Fanuc TP program (LS listing): FM144712.ls

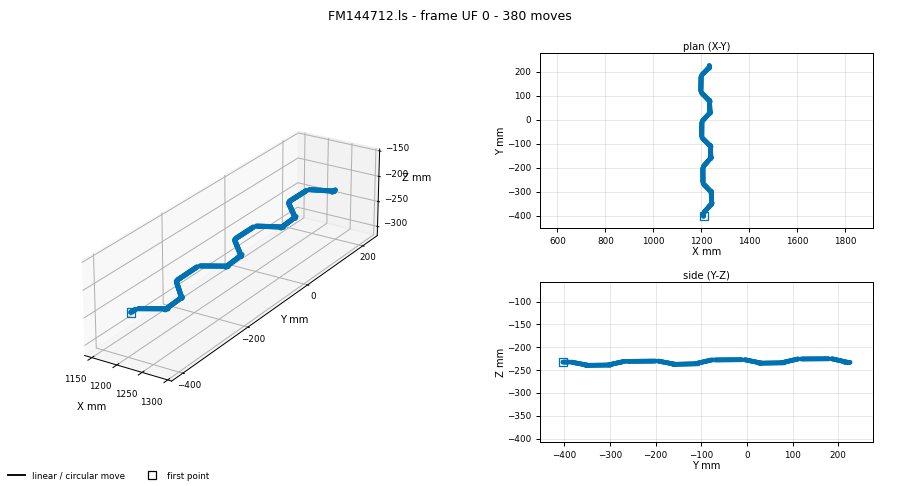
[picture p0: tool path of FM144712.ls in frame UF 0, 380 of 380 moves have a stored position in this frame; points joined in program order, loops and branches not executed]
/PROG  FM144712
/ATTR
OWNER		= MNEDITOR;
COMMENT		= "Auto FANUC move";
PROG_SIZE	= 0;
CREATE		= DATE 26-05-06  TIME 14:47:12;
MODIFIED	= DATE 26-05-06  TIME 14:47:12;
FILE_NAME	= ;
VERSION		= 0;
LINE_COUNT	= 385;
MEMORY_SIZE	= 0;
PROTECT		= READ_WRITE;
TCD:  STACK_SIZE	= 0,
      TASK_PRIORITY	= 50,
      TIME_SLICE	= 0,
      BUSY_LAMP_OFF	= 0,
      ABORT_REQUEST	= 0,
      PAUSE_REQUEST	= 0;
DEFAULT_GROUP	= 1,*,*,*,*;
CONTROL_CODE	= 00000000 00000000;
/MN
   1:  UFRAME_NUM=0 ;
   2:  UTOOL_NUM=1 ;
   3:  R[93]=10 ;
   4:  L P[1] 7mm/sec FINE ;
   5:  L P[2] 7mm/sec CNT50 ;
   6:  L P[3] 7mm/sec CNT50 ;
   7:  L P[4] 7mm/sec CNT50 ;
   8:  L P[5] 7mm/sec CNT50 ;
   9:  L P[6] 7mm/sec CNT50 ;
  10:  L P[7] 7mm/sec CNT50 ;
  11:  L P[8] 7mm/sec CNT50 ;
  12:  L P[9] 7mm/sec CNT50 ;
  13:  L P[10] 7mm/sec CNT50 ;
  14:  L P[11] 7mm/sec CNT50 ;
  15:  L P[12] 7mm/sec CNT50 ;
  16:  L P[13] 7mm/sec CNT50 ;
  17:  L P[14] 7mm/sec CNT50 ;
  18:  L P[15] 7mm/sec CNT50 ;
  19:  L P[16] 7mm/sec CNT50 ;
  20:  L P[17] 7mm/sec CNT50 ;
  21:  L P[18] 7mm/sec CNT50 ;
  22:  L P[19] 7mm/sec CNT50 ;
  23:  L P[20] 7mm/sec CNT50 ;
  24:  L P[21] 7mm/sec CNT50 ;
  25:  L P[22] 7mm/sec CNT50 ;
  26:  L P[23] 7mm/sec CNT50 ;
  27:  L P[24] 7mm/sec CNT50 ;
  28:  L P[25] 7mm/sec CNT50 ;
  29:  L P[26] 7mm/sec CNT50 ;
  30:  L P[27] 7mm/sec CNT50 ;
  31:  L P[28] 7mm/sec CNT50 ;
  32:  L P[29] 7mm/sec CNT50 ;
  33:  L P[30] 7mm/sec CNT50 ;
  34:  L P[31] 7mm/sec CNT50 ;
  35:  L P[32] 7mm/sec CNT50 ;
  36:  L P[33] 7mm/sec CNT50 ;
  37:  L P[34] 7mm/sec CNT50 ;
  38:  L P[35] 7mm/sec CNT50 ;
  39:  L P[36] 7mm/sec CNT50 ;
  40:  L P[37] 7mm/sec CNT50 ;
  41:  L P[38] 7mm/sec CNT50 ;
  42:  L P[39] 7mm/sec CNT50 ;
  43:  L P[40] 7mm/sec CNT50 ;
  44:  L P[41] 7mm/sec CNT50 ;
  45:  L P[42] 7mm/sec CNT50 ;
  46:  L P[43] 7mm/sec CNT50 ;
  47:  L P[44] 7mm/sec CNT50 ;
  48:  L P[45] 7mm/sec CNT50 ;
  49:  L P[46] 7mm/sec CNT50 ;
  50:  L P[47] 7mm/sec CNT50 ;
  51:  L P[48] 7mm/sec CNT50 ;
  52:  L P[49] 7mm/sec CNT50 ;
  53:  L P[50] 7mm/sec CNT50 ;
  54:  L P[51] 7mm/sec CNT50 ;
  55:  L P[52] 7mm/sec CNT50 ;
  56:  L P[53] 7mm/sec CNT50 ;
  57:  L P[54] 7mm/sec CNT50 ;
  58:  L P[55] 7mm/sec CNT50 ;
  59:  L P[56] 7mm/sec CNT50 ;
  60:  L P[57] 7mm/sec CNT50 ;
  61:  L P[58] 7mm/sec CNT50 ;
  62:  L P[59] 7mm/sec CNT50 ;
  63:  L P[60] 7mm/sec CNT50 ;
  64:  L P[61] 7mm/sec CNT50 ;
  65:  L P[62] 7mm/sec CNT50 ;
  66:  L P[63] 7mm/sec CNT50 ;
  67:  L P[64] 7mm/sec CNT50 ;
  68:  L P[65] 7mm/sec CNT50 ;
  69:  L P[66] 7mm/sec CNT50 ;
  70:  L P[67] 7mm/sec CNT50 ;
  71:  L P[68] 7mm/sec CNT50 ;
  72:  L P[69] 7mm/sec CNT50 ;
  73:  L P[70] 7mm/sec CNT50 ;
  74:  L P[71] 7mm/sec CNT50 ;
  75:  L P[72] 7mm/sec CNT50 ;
  76:  L P[73] 7mm/sec CNT50 ;
  77:  L P[74] 7mm/sec CNT50 ;
  78:  L P[75] 7mm/sec CNT50 ;
  79:  L P[76] 7mm/sec CNT50 ;
  80:  L P[77] 7mm/sec CNT50 ;
  81:  L P[78] 7mm/sec CNT50 ;
  82:  L P[79] 7mm/sec CNT50 ;
  83:  L P[80] 7mm/sec CNT50 ;
  84:  L P[81] 7mm/sec CNT50 ;
  85:  L P[82] 7mm/sec CNT50 ;
  86:  L P[83] 7mm/sec CNT50 ;
  87:  L P[84] 7mm/sec CNT50 ;
  88:  L P[85] 7mm/sec CNT50 ;
  89:  L P[86] 7mm/sec CNT50 ;
  90:  L P[87] 7mm/sec CNT50 ;
  91:  L P[88] 7mm/sec CNT50 ;
  92:  L P[89] 7mm/sec CNT50 ;
  93:  L P[90] 7mm/sec CNT50 ;
  94:  L P[91] 7mm/sec CNT50 ;
  95:  L P[92] 7mm/sec CNT50 ;
  96:  L P[93] 7mm/sec CNT50 ;
  97:  L P[94] 7mm/sec CNT50 ;
  98:  L P[95] 7mm/sec CNT50 ;
  99:  L P[96] 7mm/sec CNT50 ;
 100:  L P[97] 7mm/sec CNT50 ;
 101:  L P[98] 7mm/sec CNT50 ;
 102:  L P[99] 7mm/sec CNT50 ;
 103:  L P[100] 7mm/sec CNT50 ;
 104:  L P[101] 7mm/sec CNT50 ;
 105:  L P[102] 7mm/sec CNT50 ;
 106:  L P[103] 7mm/sec CNT50 ;
 107:  L P[104] 7mm/sec CNT50 ;
 108:  L P[105] 7mm/sec CNT50 ;
 109:  L P[106] 7mm/sec CNT50 ;
 110:  L P[107] 7mm/sec CNT50 ;
 111:  L P[108] 7mm/sec CNT50 ;
 112:  L P[109] 7mm/sec CNT50 ;
 113:  L P[110] 7mm/sec CNT50 ;
 114:  L P[111] 7mm/sec CNT50 ;
 115:  L P[112] 7mm/sec CNT50 ;
 116:  L P[113] 7mm/sec CNT50 ;
 117:  L P[114] 7mm/sec CNT50 ;
 118:  L P[115] 7mm/sec CNT50 ;
 119:  L P[116] 7mm/sec CNT50 ;
 120:  L P[117] 7mm/sec CNT50 ;
 121:  L P[118] 7mm/sec CNT50 ;
 122:  L P[119] 7mm/sec CNT50 ;
 123:  L P[120] 7mm/sec CNT50 ;
 124:  L P[121] 7mm/sec CNT50 ;
 125:  L P[122] 7mm/sec CNT50 ;
 126:  L P[123] 7mm/sec CNT50 ;
 127:  L P[124] 7mm/sec CNT50 ;
 128:  L P[125] 7mm/sec CNT50 ;
 129:  L P[126] 7mm/sec CNT50 ;
 130:  L P[127] 7mm/sec CNT50 ;
 131:  L P[128] 7mm/sec CNT50 ;
 132:  L P[129] 7mm/sec CNT50 ;
 133:  L P[130] 7mm/sec CNT50 ;
 134:  L P[131] 7mm/sec CNT50 ;
 135:  L P[132] 7mm/sec CNT50 ;
 136:  L P[133] 7mm/sec CNT50 ;
 137:  L P[134] 7mm/sec CNT50 ;
 138:  L P[135] 7mm/sec CNT50 ;
 139:  L P[136] 7mm/sec CNT50 ;
 140:  L P[137] 7mm/sec CNT50 ;
 141:  L P[138] 7mm/sec CNT50 ;
 142:  L P[139] 7mm/sec CNT50 ;
 143:  L P[140] 7mm/sec CNT50 ;
 144:  L P[141] 7mm/sec CNT50 ;
 145:  L P[142] 7mm/sec CNT50 ;
 146:  L P[143] 7mm/sec CNT50 ;
 147:  L P[144] 7mm/sec CNT50 ;
 148:  L P[145] 7mm/sec CNT50 ;
 149:  L P[146] 7mm/sec CNT50 ;
 150:  L P[147] 7mm/sec CNT50 ;
 151:  L P[148] 7mm/sec CNT50 ;
 152:  L P[149] 7mm/sec CNT50 ;
 153:  L P[150] 7mm/sec CNT50 ;
 154:  L P[151] 7mm/sec CNT50 ;
 155:  L P[152] 7mm/sec CNT50 ;
 156:  L P[153] 7mm/sec CNT50 ;
 157:  L P[154] 7mm/sec CNT50 ;
 158:  L P[155] 7mm/sec CNT50 ;
 159:  L P[156] 7mm/sec CNT50 ;
 160:  L P[157] 7mm/sec CNT50 ;
 161:  L P[158] 7mm/sec CNT50 ;
 162:  L P[159] 7mm/sec CNT50 ;
 163:  L P[160] 7mm/sec CNT50 ;
 164:  L P[161] 7mm/sec CNT50 ;
 165:  L P[162] 7mm/sec CNT50 ;
 166:  L P[163] 7mm/sec CNT50 ;
 167:  L P[164] 7mm/sec CNT50 ;
 168:  L P[165] 7mm/sec CNT50 ;
 169:  L P[166] 7mm/sec CNT50 ;
 170:  L P[167] 7mm/sec CNT50 ;
 171:  L P[168] 7mm/sec CNT50 ;
 172:  L P[169] 7mm/sec CNT50 ;
 173:  L P[170] 7mm/sec CNT50 ;
 174:  L P[171] 7mm/sec CNT50 ;
 175:  L P[172] 7mm/sec CNT50 ;
 176:  L P[173] 7mm/sec CNT50 ;
 177:  L P[174] 7mm/sec CNT50 ;
 178:  L P[175] 7mm/sec CNT50 ;
 179:  L P[176] 7mm/sec CNT50 ;
 180:  L P[177] 7mm/sec CNT50 ;
 181:  L P[178] 7mm/sec CNT50 ;
 182:  L P[179] 7mm/sec CNT50 ;
 183:  L P[180] 7mm/sec CNT50 ;
 184:  L P[181] 7mm/sec CNT50 ;
 185:  L P[182] 7mm/sec CNT50 ;
 186:  L P[183] 7mm/sec CNT50 ;
 187:  L P[184] 7mm/sec CNT50 ;
 188:  L P[185] 7mm/sec CNT50 ;
 189:  L P[186] 7mm/sec CNT50 ;
 190:  L P[187] 7mm/sec CNT50 ;
 191:  L P[188] 7mm/sec CNT50 ;
 192:  L P[189] 7mm/sec CNT50 ;
 193:  L P[190] 7mm/sec CNT50 ;
 194:  L P[191] 7mm/sec CNT50 ;
 195:  L P[192] 7mm/sec CNT50 ;
 196:  L P[193] 7mm/sec CNT50 ;
 197:  L P[194] 7mm/sec CNT50 ;
 198:  L P[195] 7mm/sec CNT50 ;
 199:  L P[196] 7mm/sec CNT50 ;
 200:  L P[197] 7mm/sec CNT50 ;
 201:  L P[198] 7mm/sec CNT50 ;
 202:  L P[199] 7mm/sec CNT50 ;
 203:  L P[200] 7mm/sec CNT50 ;
 204:  L P[201] 7mm/sec CNT50 ;
 205:  L P[202] 7mm/sec CNT50 ;
 206:  L P[203] 7mm/sec CNT50 ;
 207:  L P[204] 7mm/sec CNT50 ;
 208:  L P[205] 7mm/sec CNT50 ;
 209:  L P[206] 7mm/sec CNT50 ;
 210:  L P[207] 7mm/sec CNT50 ;
 211:  L P[208] 7mm/sec CNT50 ;
 212:  L P[209] 7mm/sec CNT50 ;
 213:  L P[210] 7mm/sec CNT50 ;
 214:  L P[211] 7mm/sec CNT50 ;
 215:  L P[212] 7mm/sec CNT50 ;
 216:  L P[213] 7mm/sec CNT50 ;
 217:  L P[214] 7mm/sec CNT50 ;
 218:  L P[215] 7mm/sec CNT50 ;
 219:  L P[216] 7mm/sec CNT50 ;
 220:  L P[217] 7mm/sec CNT50 ;
 221:  L P[218] 7mm/sec CNT50 ;
 222:  L P[219] 7mm/sec CNT50 ;
 223:  L P[220] 7mm/sec CNT50 ;
 224:  L P[221] 7mm/sec CNT50 ;
 225:  L P[222] 7mm/sec CNT50 ;
 226:  L P[223] 7mm/sec CNT50 ;
 227:  L P[224] 7mm/sec CNT50 ;
 228:  L P[225] 7mm/sec CNT50 ;
 229:  L P[226] 7mm/sec CNT50 ;
 230:  L P[227] 7mm/sec CNT50 ;
 231:  L P[228] 7mm/sec CNT50 ;
 232:  L P[229] 7mm/sec CNT50 ;
 233:  L P[230] 7mm/sec CNT50 ;
 234:  L P[231] 7mm/sec CNT50 ;
 235:  L P[232] 7mm/sec CNT50 ;
 236:  L P[233] 7mm/sec CNT50 ;
 237:  L P[234] 7mm/sec CNT50 ;
 238:  L P[235] 7mm/sec CNT50 ;
 239:  L P[236] 7mm/sec CNT50 ;
 240:  L P[237] 7mm/sec CNT50 ;
 241:  L P[238] 7mm/sec CNT50 ;
 242:  L P[239] 7mm/sec CNT50 ;
 243:  L P[240] 7mm/sec CNT50 ;
 244:  L P[241] 7mm/sec CNT50 ;
 245:  L P[242] 7mm/sec CNT50 ;
 246:  L P[243] 7mm/sec CNT50 ;
 247:  L P[244] 7mm/sec CNT50 ;
 248:  L P[245] 7mm/sec CNT50 ;
 249:  L P[246] 7mm/sec CNT50 ;
 250:  L P[247] 7mm/sec CNT50 ;
 251:  L P[248] 7mm/sec CNT50 ;
 252:  L P[249] 7mm/sec CNT50 ;
 253:  L P[250] 7mm/sec CNT50 ;
 254:  L P[251] 7mm/sec CNT50 ;
 255:  L P[252] 7mm/sec CNT50 ;
 256:  L P[253] 7mm/sec CNT50 ;
 257:  L P[254] 7mm/sec CNT50 ;
 258:  L P[255] 7mm/sec CNT50 ;
 259:  L P[256] 7mm/sec CNT50 ;
 260:  L P[257] 7mm/sec CNT50 ;
 261:  L P[258] 7mm/sec CNT50 ;
 262:  L P[259] 7mm/sec CNT50 ;
 263:  L P[260] 7mm/sec CNT50 ;
 264:  L P[261] 7mm/sec CNT50 ;
 265:  L P[262] 7mm/sec CNT50 ;
 266:  L P[263] 7mm/sec CNT50 ;
 267:  L P[264] 7mm/sec CNT50 ;
 268:  L P[265] 7mm/sec CNT50 ;
 269:  L P[266] 7mm/sec CNT50 ;
 270:  L P[267] 7mm/sec CNT50 ;
 271:  L P[268] 7mm/sec CNT50 ;
 272:  L P[269] 7mm/sec CNT50 ;
 273:  L P[270] 7mm/sec CNT50 ;
 274:  L P[271] 7mm/sec CNT50 ;
 275:  L P[272] 7mm/sec CNT50 ;
 276:  L P[273] 7mm/sec CNT50 ;
 277:  L P[274] 7mm/sec CNT50 ;
 278:  L P[275] 7mm/sec CNT50 ;
 279:  L P[276] 7mm/sec CNT50 ;
 280:  L P[277] 7mm/sec CNT50 ;
 281:  L P[278] 7mm/sec CNT50 ;
 282:  L P[279] 7mm/sec CNT50 ;
 283:  L P[280] 7mm/sec CNT50 ;
 284:  L P[281] 7mm/sec CNT50 ;
 285:  L P[282] 7mm/sec CNT50 ;
 286:  L P[283] 7mm/sec CNT50 ;
 287:  L P[284] 7mm/sec CNT50 ;
 288:  L P[285] 7mm/sec CNT50 ;
 289:  L P[286] 7mm/sec CNT50 ;
 290:  L P[287] 7mm/sec CNT50 ;
 291:  L P[288] 7mm/sec CNT50 ;
 292:  L P[289] 7mm/sec CNT50 ;
 293:  L P[290] 7mm/sec CNT50 ;
 294:  L P[291] 7mm/sec CNT50 ;
 295:  L P[292] 7mm/sec CNT50 ;
 296:  L P[293] 7mm/sec CNT50 ;
 297:  L P[294] 7mm/sec CNT50 ;
 298:  L P[295] 7mm/sec CNT50 ;
 299:  L P[296] 7mm/sec CNT50 ;
 300:  L P[297] 7mm/sec CNT50 ;
 301:  L P[298] 7mm/sec CNT50 ;
 302:  L P[299] 7mm/sec CNT50 ;
 303:  L P[300] 7mm/sec CNT50 ;
 304:  L P[301] 7mm/sec CNT50 ;
 305:  L P[302] 7mm/sec CNT50 ;
 306:  L P[303] 7mm/sec CNT50 ;
 307:  L P[304] 7mm/sec CNT50 ;
 308:  L P[305] 7mm/sec CNT50 ;
 309:  L P[306] 7mm/sec CNT50 ;
 310:  L P[307] 7mm/sec CNT50 ;
 311:  L P[308] 7mm/sec CNT50 ;
 312:  L P[309] 7mm/sec CNT50 ;
 313:  L P[310] 7mm/sec CNT50 ;
 314:  L P[311] 7mm/sec CNT50 ;
 315:  L P[312] 7mm/sec CNT50 ;
 316:  L P[313] 7mm/sec CNT50 ;
 317:  L P[314] 7mm/sec CNT50 ;
 318:  L P[315] 7mm/sec CNT50 ;
 319:  L P[316] 7mm/sec CNT50 ;
 320:  L P[317] 7mm/sec CNT50 ;
 321:  L P[318] 7mm/sec CNT50 ;
 322:  L P[319] 7mm/sec CNT50 ;
 323:  L P[320] 7mm/sec CNT50 ;
 324:  L P[321] 7mm/sec CNT50 ;
 325:  L P[322] 7mm/sec CNT50 ;
 326:  L P[323] 7mm/sec CNT50 ;
 327:  L P[324] 7mm/sec CNT50 ;
 328:  L P[325] 7mm/sec CNT50 ;
 329:  L P[326] 7mm/sec CNT50 ;
 330:  L P[327] 7mm/sec CNT50 ;
 331:  L P[328] 7mm/sec CNT50 ;
 332:  L P[329] 7mm/sec CNT50 ;
 333:  L P[330] 7mm/sec CNT50 ;
 334:  L P[331] 7mm/sec CNT50 ;
 335:  L P[332] 7mm/sec CNT50 ;
 336:  L P[333] 7mm/sec CNT50 ;
 337:  L P[334] 7mm/sec CNT50 ;
 338:  L P[335] 7mm/sec CNT50 ;
 339:  L P[336] 7mm/sec CNT50 ;
 340:  L P[337] 7mm/sec CNT50 ;
 341:  L P[338] 7mm/sec CNT50 ;
 342:  L P[339] 7mm/sec CNT50 ;
 343:  L P[340] 7mm/sec CNT50 ;
 344:  L P[341] 7mm/sec CNT50 ;
 345:  L P[342] 7mm/sec CNT50 ;
 346:  L P[343] 7mm/sec CNT50 ;
 347:  L P[344] 7mm/sec CNT50 ;
 348:  L P[345] 7mm/sec CNT50 ;
 349:  L P[346] 7mm/sec CNT50 ;
 350:  L P[347] 7mm/sec CNT50 ;
 351:  L P[348] 7mm/sec CNT50 ;
 352:  L P[349] 7mm/sec CNT50 ;
 353:  L P[350] 7mm/sec CNT50 ;
 354:  L P[351] 7mm/sec CNT50 ;
 355:  L P[352] 7mm/sec CNT50 ;
 356:  L P[353] 7mm/sec CNT50 ;
 357:  L P[354] 7mm/sec CNT50 ;
 358:  L P[355] 7mm/sec CNT50 ;
 359:  L P[356] 7mm/sec CNT50 ;
 360:  L P[357] 7mm/sec CNT50 ;
 361:  L P[358] 7mm/sec CNT50 ;
 362:  L P[359] 7mm/sec CNT50 ;
 363:  L P[360] 7mm/sec CNT50 ;
 364:  L P[361] 7mm/sec CNT50 ;
 365:  L P[362] 7mm/sec CNT50 ;
 366:  L P[363] 7mm/sec CNT50 ;
 367:  L P[364] 7mm/sec CNT50 ;
 368:  L P[365] 7mm/sec CNT50 ;
 369:  L P[366] 7mm/sec CNT50 ;
 370:  L P[367] 7mm/sec CNT50 ;
 371:  L P[368] 7mm/sec CNT50 ;
 372:  L P[369] 7mm/sec CNT50 ;
 373:  L P[370] 7mm/sec CNT50 ;
 374:  L P[371] 7mm/sec CNT50 ;
 375:  L P[372] 7mm/sec CNT50 ;
 376:  L P[373] 7mm/sec CNT50 ;
 377:  L P[374] 7mm/sec CNT50 ;
 378:  L P[375] 7mm/sec CNT50 ;
 379:  L P[376] 7mm/sec CNT50 ;
 380:  L P[377] 7mm/sec CNT50 ;
 381:  L P[378] 7mm/sec CNT50 ;
 382:  L P[379] 7mm/sec CNT50 ;
 383:  L P[380] 7mm/sec FINE ;
 384:  R[93]=1 ;
 385:  END ;
/POS
P[1]{
   GP1:
	UF : 0, UT : 1,		CONFIG : 'N U T, 0, 0, 0',
	X = 1209.451  mm,	Y = -403.216  mm,	Z = -232.520  mm,
	W = 0.000 deg,	P = 30.000 deg,	R = 178.127 deg
};
P[2]{
   GP1:
	UF : 0, UT : 1,		CONFIG : 'N U T, 0, 0, 0',
	X = 1209.517  mm,	Y = -401.217  mm,	Z = -232.512  mm,
	W = 0.000 deg,	P = 30.000 deg,	R = 178.127 deg
};
P[3]{
   GP1:
	UF : 0, UT : 1,		CONFIG : 'N U T, 0, 0, 0',
	X = 1209.582  mm,	Y = -399.218  mm,	Z = -232.503  mm,
	W = 0.000 deg,	P = 30.000 deg,	R = 170.876 deg
};
P[4]{
   GP1:
	UF : 0, UT : 1,		CONFIG : 'N U T, 0, 0, 0',
	X = 1209.647  mm,	Y = -397.220  mm,	Z = -232.495  mm,
	W = 0.000 deg,	P = 30.000 deg,	R = 167.251 deg
};
P[5]{
   GP1:
	UF : 0, UT : 1,		CONFIG : 'N U T, 0, 0, 0',
	X = 1209.713  mm,	Y = -395.221  mm,	Z = -232.486  mm,
	W = 0.000 deg,	P = 30.000 deg,	R = 163.625 deg
};
P[6]{
   GP1:
	UF : 0, UT : 1,		CONFIG : 'N U T, 0, 0, 0',
	X = 1209.778  mm,	Y = -393.222  mm,	Z = -232.478  mm,
	W = 0.000 deg,	P = 30.000 deg,	R = 160.000 deg
};
P[7]{
   GP1:
	UF : 0, UT : 1,		CONFIG : 'N U T, 0, 0, 0',
	X = 1209.922  mm,	Y = -390.499  mm,	Z = -232.471  mm,
	W = 0.000 deg,	P = 30.000 deg,	R = 160.000 deg
};
P[8]{
   GP1:
	UF : 0, UT : 1,		CONFIG : 'N U T, 0, 0, 0',
	X = 1212.525  mm,	Y = -385.034  mm,	Z = -232.516  mm,
	W = 0.000 deg,	P = 30.000 deg,	R = 160.000 deg
};
P[9]{
   GP1:
	UF : 0, UT : 1,		CONFIG : 'N U T, 0, 0, 0',
	X = 1213.831  mm,	Y = -383.546  mm,	Z = -232.798  mm,
	W = 0.000 deg,	P = 30.000 deg,	R = 160.000 deg
};
P[10]{
   GP1:
	UF : 0, UT : 1,		CONFIG : 'N U T, 0, 0, 0',
	X = 1215.138  mm,	Y = -382.058  mm,	Z = -233.080  mm,
	W = 0.000 deg,	P = 30.000 deg,	R = 160.000 deg
};
P[11]{
   GP1:
	UF : 0, UT : 1,		CONFIG : 'N U T, 0, 0, 0',
	X = 1216.444  mm,	Y = -380.570  mm,	Z = -233.362  mm,
	W = 0.000 deg,	P = 30.000 deg,	R = 160.000 deg
};
P[12]{
   GP1:
	UF : 0, UT : 1,		CONFIG : 'N U T, 0, 0, 0',
	X = 1217.751  mm,	Y = -379.082  mm,	Z = -233.644  mm,
	W = 0.000 deg,	P = 30.000 deg,	R = 160.000 deg
};
P[13]{
   GP1:
	UF : 0, UT : 1,		CONFIG : 'N U T, 0, 0, 0',
	X = 1219.057  mm,	Y = -377.595  mm,	Z = -233.926  mm,
	W = 0.000 deg,	P = 30.000 deg,	R = 160.000 deg
};
P[14]{
   GP1:
	UF : 0, UT : 1,		CONFIG : 'N U T, 0, 0, 0',
	X = 1220.364  mm,	Y = -376.107  mm,	Z = -234.208  mm,
	W = 0.000 deg,	P = 30.000 deg,	R = 160.000 deg
};
P[15]{
   GP1:
	UF : 0, UT : 1,		CONFIG : 'N U T, 0, 0, 0',
	X = 1221.670  mm,	Y = -374.619  mm,	Z = -234.490  mm,
	W = 0.000 deg,	P = 30.000 deg,	R = 160.000 deg
};
P[16]{
   GP1:
	UF : 0, UT : 1,		CONFIG : 'N U T, 0, 0, 0',
	X = 1222.977  mm,	Y = -373.131  mm,	Z = -234.772  mm,
	W = 0.000 deg,	P = 30.000 deg,	R = 160.000 deg
};
P[17]{
   GP1:
	UF : 0, UT : 1,		CONFIG : 'N U T, 0, 0, 0',
	X = 1224.283  mm,	Y = -371.644  mm,	Z = -235.054  mm,
	W = 0.000 deg,	P = 30.000 deg,	R = 160.000 deg
};
P[18]{
   GP1:
	UF : 0, UT : 1,		CONFIG : 'N U T, 0, 0, 0',
	X = 1225.590  mm,	Y = -370.156  mm,	Z = -235.336  mm,
	W = 0.000 deg,	P = 30.000 deg,	R = 160.000 deg
};
P[19]{
   GP1:
	UF : 0, UT : 1,		CONFIG : 'N U T, 0, 0, 0',
	X = 1226.896  mm,	Y = -368.668  mm,	Z = -235.618  mm,
	W = 0.000 deg,	P = 30.000 deg,	R = 160.000 deg
};
P[20]{
   GP1:
	UF : 0, UT : 1,		CONFIG : 'N U T, 0, 0, 0',
	X = 1228.203  mm,	Y = -367.180  mm,	Z = -235.900  mm,
	W = 0.000 deg,	P = 30.000 deg,	R = 160.000 deg
};
P[21]{
   GP1:
	UF : 0, UT : 1,		CONFIG : 'N U T, 0, 0, 0',
	X = 1229.510  mm,	Y = -365.692  mm,	Z = -236.181  mm,
	W = 0.000 deg,	P = 30.000 deg,	R = 160.000 deg
};
P[22]{
   GP1:
	UF : 0, UT : 1,		CONFIG : 'N U T, 0, 0, 0',
	X = 1230.816  mm,	Y = -364.205  mm,	Z = -236.463  mm,
	W = 0.000 deg,	P = 30.000 deg,	R = 160.000 deg
};
P[23]{
   GP1:
	UF : 0, UT : 1,		CONFIG : 'N U T, 0, 0, 0',
	X = 1232.123  mm,	Y = -362.717  mm,	Z = -236.745  mm,
	W = 0.000 deg,	P = 30.000 deg,	R = 160.000 deg
};
P[24]{
   GP1:
	UF : 0, UT : 1,		CONFIG : 'N U T, 0, 0, 0',
	X = 1233.429  mm,	Y = -361.229  mm,	Z = -237.027  mm,
	W = 0.000 deg,	P = 30.000 deg,	R = 160.000 deg
};
P[25]{
   GP1:
	UF : 0, UT : 1,		CONFIG : 'N U T, 0, 0, 0',
	X = 1234.736  mm,	Y = -359.741  mm,	Z = -237.309  mm,
	W = 0.000 deg,	P = 30.000 deg,	R = 160.000 deg
};
P[26]{
   GP1:
	UF : 0, UT : 1,		CONFIG : 'N U T, 0, 0, 0',
	X = 1236.042  mm,	Y = -358.253  mm,	Z = -237.591  mm,
	W = 0.000 deg,	P = 30.000 deg,	R = 160.000 deg
};
P[27]{
   GP1:
	UF : 0, UT : 1,		CONFIG : 'N U T, 0, 0, 0',
	X = 1237.349  mm,	Y = -356.766  mm,	Z = -237.873  mm,
	W = 0.000 deg,	P = 30.000 deg,	R = 160.000 deg
};
P[28]{
   GP1:
	UF : 0, UT : 1,		CONFIG : 'N U T, 0, 0, 0',
	X = 1238.655  mm,	Y = -355.278  mm,	Z = -238.155  mm,
	W = 0.000 deg,	P = 30.000 deg,	R = 160.000 deg
};
P[29]{
   GP1:
	UF : 0, UT : 1,		CONFIG : 'N U T, 0, 0, 0',
	X = 1239.962  mm,	Y = -353.790  mm,	Z = -238.437  mm,
	W = 0.000 deg,	P = 30.000 deg,	R = 165.095 deg
};
P[30]{
   GP1:
	UF : 0, UT : 1,		CONFIG : 'N U T, 0, 0, 0',
	X = 1241.268  mm,	Y = -352.302  mm,	Z = -238.719  mm,
	W = 0.000 deg,	P = 30.000 deg,	R = 169.481 deg
};
P[31]{
   GP1:
	UF : 0, UT : 1,		CONFIG : 'N U T, 0, 0, 0',
	X = 1242.575  mm,	Y = -350.815  mm,	Z = -239.001  mm,
	W = 0.000 deg,	P = 30.000 deg,	R = 173.867 deg
};
P[32]{
   GP1:
	UF : 0, UT : 1,		CONFIG : 'N U T, 0, 0, 0',
	X = 1243.881  mm,	Y = -349.327  mm,	Z = -239.283  mm,
	W = 0.000 deg,	P = 30.000 deg,	R = 178.253 deg
};
P[33]{
   GP1:
	UF : 0, UT : 1,		CONFIG : 'N U T, 0, 0, 0',
	X = 1245.188  mm,	Y = -347.839  mm,	Z = -239.565  mm,
	W = 0.000 deg,	P = 30.000 deg,	R = -178.069 deg
};
P[34]{
   GP1:
	UF : 0, UT : 1,		CONFIG : 'N U T, 0, 0, 0',
	X = 1243.047  mm,	Y = -352.949  mm,	Z = -239.624  mm,
	W = 0.000 deg,	P = 30.000 deg,	R = -178.069 deg
};
P[35]{
   GP1:
	UF : 0, UT : 1,		CONFIG : 'N U T, 0, 0, 0',
	X = 1242.931  mm,	Y = -352.884  mm,	Z = -239.602  mm,
	W = 0.000 deg,	P = 30.000 deg,	R = -178.069 deg
};
P[36]{
   GP1:
	UF : 0, UT : 1,		CONFIG : 'N U T, 0, 0, 0',
	X = 1242.864  mm,	Y = -350.885  mm,	Z = -239.574  mm,
	W = 0.000 deg,	P = 30.000 deg,	R = -178.069 deg
};
P[37]{
   GP1:
	UF : 0, UT : 1,		CONFIG : 'N U T, 0, 0, 0',
	X = 1242.796  mm,	Y = -348.887  mm,	Z = -239.545  mm,
	W = 0.000 deg,	P = 30.000 deg,	R = -178.069 deg
};
P[38]{
   GP1:
	UF : 0, UT : 1,		CONFIG : 'N U T, 0, 0, 0',
	X = 1242.729  mm,	Y = -346.888  mm,	Z = -239.517  mm,
	W = 0.000 deg,	P = 30.000 deg,	R = -178.069 deg
};
P[39]{
   GP1:
	UF : 0, UT : 1,		CONFIG : 'N U T, 0, 0, 0',
	X = 1242.661  mm,	Y = -344.889  mm,	Z = -239.489  mm,
	W = 0.000 deg,	P = 30.000 deg,	R = -178.069 deg
};
P[40]{
   GP1:
	UF : 0, UT : 1,		CONFIG : 'N U T, 0, 0, 0',
	X = 1242.594  mm,	Y = -342.891  mm,	Z = -239.460  mm,
	W = 0.000 deg,	P = 30.000 deg,	R = -178.069 deg
};
P[41]{
   GP1:
	UF : 0, UT : 1,		CONFIG : 'N U T, 0, 0, 0',
	X = 1242.527  mm,	Y = -340.892  mm,	Z = -239.432  mm,
	W = 0.000 deg,	P = 30.000 deg,	R = -178.069 deg
};
P[42]{
   GP1:
	UF : 0, UT : 1,		CONFIG : 'N U T, 0, 0, 0',
	X = 1242.459  mm,	Y = -338.893  mm,	Z = -239.404  mm,
	W = 0.000 deg,	P = 30.000 deg,	R = -178.069 deg
};
P[43]{
   GP1:
	UF : 0, UT : 1,		CONFIG : 'N U T, 0, 0, 0',
	X = 1242.392  mm,	Y = -336.895  mm,	Z = -239.375  mm,
	W = 0.000 deg,	P = 30.000 deg,	R = -178.069 deg
};
P[44]{
   GP1:
	UF : 0, UT : 1,		CONFIG : 'N U T, 0, 0, 0',
	X = 1242.324  mm,	Y = -334.896  mm,	Z = -239.347  mm,
	W = 0.000 deg,	P = 30.000 deg,	R = -178.069 deg
};
P[45]{
   GP1:
	UF : 0, UT : 1,		CONFIG : 'N U T, 0, 0, 0',
	X = 1242.257  mm,	Y = -332.897  mm,	Z = -239.319  mm,
	W = 0.000 deg,	P = 30.000 deg,	R = -178.069 deg
};
P[46]{
   GP1:
	UF : 0, UT : 1,		CONFIG : 'N U T, 0, 0, 0',
	X = 1242.190  mm,	Y = -330.899  mm,	Z = -239.290  mm,
	W = 0.000 deg,	P = 30.000 deg,	R = -178.069 deg
};
P[47]{
   GP1:
	UF : 0, UT : 1,		CONFIG : 'N U T, 0, 0, 0',
	X = 1242.122  mm,	Y = -328.900  mm,	Z = -239.262  mm,
	W = 0.000 deg,	P = 30.000 deg,	R = -178.069 deg
};
P[48]{
   GP1:
	UF : 0, UT : 1,		CONFIG : 'N U T, 0, 0, 0',
	X = 1242.055  mm,	Y = -326.901  mm,	Z = -239.234  mm,
	W = 0.000 deg,	P = 30.000 deg,	R = -178.069 deg
};
P[49]{
   GP1:
	UF : 0, UT : 1,		CONFIG : 'N U T, 0, 0, 0',
	X = 1241.988  mm,	Y = -324.903  mm,	Z = -239.205  mm,
	W = 0.000 deg,	P = 30.000 deg,	R = -178.069 deg
};
P[50]{
   GP1:
	UF : 0, UT : 1,		CONFIG : 'N U T, 0, 0, 0',
	X = 1241.920  mm,	Y = -322.904  mm,	Z = -239.177  mm,
	W = 0.000 deg,	P = 30.000 deg,	R = -178.069 deg
};
P[51]{
   GP1:
	UF : 0, UT : 1,		CONFIG : 'N U T, 0, 0, 0',
	X = 1241.853  mm,	Y = -320.905  mm,	Z = -239.149  mm,
	W = 0.000 deg,	P = 30.000 deg,	R = -178.069 deg
};
P[52]{
   GP1:
	UF : 0, UT : 1,		CONFIG : 'N U T, 0, 0, 0',
	X = 1241.785  mm,	Y = -318.907  mm,	Z = -239.120  mm,
	W = 0.000 deg,	P = 30.000 deg,	R = -178.069 deg
};
P[53]{
   GP1:
	UF : 0, UT : 1,		CONFIG : 'N U T, 0, 0, 0',
	X = 1241.718  mm,	Y = -316.908  mm,	Z = -239.092  mm,
	W = 0.000 deg,	P = 30.000 deg,	R = -178.069 deg
};
P[54]{
   GP1:
	UF : 0, UT : 1,		CONFIG : 'N U T, 0, 0, 0',
	X = 1241.651  mm,	Y = -314.909  mm,	Z = -239.064  mm,
	W = 0.000 deg,	P = 30.000 deg,	R = -178.069 deg
};
P[55]{
   GP1:
	UF : 0, UT : 1,		CONFIG : 'N U T, 0, 0, 0',
	X = 1241.583  mm,	Y = -312.911  mm,	Z = -239.035  mm,
	W = 0.000 deg,	P = 30.000 deg,	R = -178.069 deg
};
P[56]{
   GP1:
	UF : 0, UT : 1,		CONFIG : 'N U T, 0, 0, 0',
	X = 1241.516  mm,	Y = -310.912  mm,	Z = -239.007  mm,
	W = 0.000 deg,	P = 30.000 deg,	R = -178.069 deg
};
P[57]{
   GP1:
	UF : 0, UT : 1,		CONFIG : 'N U T, 0, 0, 0',
	X = 1241.448  mm,	Y = -308.913  mm,	Z = -238.979  mm,
	W = 0.000 deg,	P = 30.000 deg,	R = -178.069 deg
};
P[58]{
   GP1:
	UF : 0, UT : 1,		CONFIG : 'N U T, 0, 0, 0',
	X = 1241.381  mm,	Y = -306.915  mm,	Z = -238.950  mm,
	W = 0.000 deg,	P = 30.000 deg,	R = -178.069 deg
};
P[59]{
   GP1:
	UF : 0, UT : 1,		CONFIG : 'N U T, 0, 0, 0',
	X = 1241.314  mm,	Y = -304.916  mm,	Z = -238.922  mm,
	W = 0.000 deg,	P = 30.000 deg,	R = -171.606 deg
};
P[60]{
   GP1:
	UF : 0, UT : 1,		CONFIG : 'N U T, 0, 0, 0',
	X = 1241.246  mm,	Y = -302.917  mm,	Z = -238.893  mm,
	W = 0.000 deg,	P = 30.000 deg,	R = -167.993 deg
};
P[61]{
   GP1:
	UF : 0, UT : 1,		CONFIG : 'N U T, 0, 0, 0',
	X = 1241.179  mm,	Y = -300.919  mm,	Z = -238.865  mm,
	W = 0.000 deg,	P = 30.000 deg,	R = -164.379 deg
};
P[62]{
   GP1:
	UF : 0, UT : 1,		CONFIG : 'N U T, 0, 0, 0',
	X = 1241.112  mm,	Y = -298.920  mm,	Z = -238.837  mm,
	W = 0.000 deg,	P = 30.000 deg,	R = -160.765 deg
};
P[63]{
   GP1:
	UF : 0, UT : 1,		CONFIG : 'N U T, 0, 0, 0',
	X = 1241.493  mm,	Y = -300.213  mm,	Z = -238.819  mm,
	W = 0.000 deg,	P = 30.000 deg,	R = -160.000 deg
};
P[64]{
   GP1:
	UF : 0, UT : 1,		CONFIG : 'N U T, 0, 0, 0',
	X = 1243.361  mm,	Y = -303.731  mm,	Z = -238.703  mm,
	W = 0.000 deg,	P = 30.000 deg,	R = -160.000 deg
};
P[65]{
   GP1:
	UF : 0, UT : 1,		CONFIG : 'N U T, 0, 0, 0',
	X = 1241.991  mm,	Y = -302.309  mm,	Z = -238.384  mm,
	W = 0.000 deg,	P = 30.000 deg,	R = -160.000 deg
};
P[66]{
   GP1:
	UF : 0, UT : 1,		CONFIG : 'N U T, 0, 0, 0',
	X = 1240.622  mm,	Y = -300.887  mm,	Z = -238.065  mm,
	W = 0.000 deg,	P = 30.000 deg,	R = -160.000 deg
};
P[67]{
   GP1:
	UF : 0, UT : 1,		CONFIG : 'N U T, 0, 0, 0',
	X = 1239.252  mm,	Y = -299.465  mm,	Z = -237.747  mm,
	W = 0.000 deg,	P = 30.000 deg,	R = -160.000 deg
};
P[68]{
   GP1:
	UF : 0, UT : 1,		CONFIG : 'N U T, 0, 0, 0',
	X = 1237.882  mm,	Y = -298.042  mm,	Z = -237.428  mm,
	W = 0.000 deg,	P = 30.000 deg,	R = -160.000 deg
};
P[69]{
   GP1:
	UF : 0, UT : 1,		CONFIG : 'N U T, 0, 0, 0',
	X = 1236.513  mm,	Y = -296.620  mm,	Z = -237.110  mm,
	W = 0.000 deg,	P = 30.000 deg,	R = -160.000 deg
};
P[70]{
   GP1:
	UF : 0, UT : 1,		CONFIG : 'N U T, 0, 0, 0',
	X = 1235.143  mm,	Y = -295.198  mm,	Z = -236.791  mm,
	W = 0.000 deg,	P = 30.000 deg,	R = -160.000 deg
};
P[71]{
   GP1:
	UF : 0, UT : 1,		CONFIG : 'N U T, 0, 0, 0',
	X = 1233.774  mm,	Y = -293.776  mm,	Z = -236.472  mm,
	W = 0.000 deg,	P = 30.000 deg,	R = -160.000 deg
};
P[72]{
   GP1:
	UF : 0, UT : 1,		CONFIG : 'N U T, 0, 0, 0',
	X = 1232.404  mm,	Y = -292.354  mm,	Z = -236.154  mm,
	W = 0.000 deg,	P = 30.000 deg,	R = -160.000 deg
};
P[73]{
   GP1:
	UF : 0, UT : 1,		CONFIG : 'N U T, 0, 0, 0',
	X = 1231.034  mm,	Y = -290.931  mm,	Z = -235.835  mm,
	W = 0.000 deg,	P = 30.000 deg,	R = -160.000 deg
};
P[74]{
   GP1:
	UF : 0, UT : 1,		CONFIG : 'N U T, 0, 0, 0',
	X = 1229.665  mm,	Y = -289.509  mm,	Z = -235.516  mm,
	W = 0.000 deg,	P = 30.000 deg,	R = -160.000 deg
};
P[75]{
   GP1:
	UF : 0, UT : 1,		CONFIG : 'N U T, 0, 0, 0',
	X = 1228.295  mm,	Y = -288.087  mm,	Z = -235.198  mm,
	W = 0.000 deg,	P = 30.000 deg,	R = -160.000 deg
};
P[76]{
   GP1:
	UF : 0, UT : 1,		CONFIG : 'N U T, 0, 0, 0',
	X = 1226.926  mm,	Y = -286.665  mm,	Z = -234.879  mm,
	W = 0.000 deg,	P = 30.000 deg,	R = -160.000 deg
};
P[77]{
   GP1:
	UF : 0, UT : 1,		CONFIG : 'N U T, 0, 0, 0',
	X = 1225.556  mm,	Y = -285.243  mm,	Z = -234.561  mm,
	W = 0.000 deg,	P = 30.000 deg,	R = -160.000 deg
};
P[78]{
   GP1:
	UF : 0, UT : 1,		CONFIG : 'N U T, 0, 0, 0',
	X = 1224.186  mm,	Y = -283.820  mm,	Z = -234.242  mm,
	W = 0.000 deg,	P = 30.000 deg,	R = -160.000 deg
};
P[79]{
   GP1:
	UF : 0, UT : 1,		CONFIG : 'N U T, 0, 0, 0',
	X = 1222.817  mm,	Y = -282.398  mm,	Z = -233.923  mm,
	W = 0.000 deg,	P = 30.000 deg,	R = -160.000 deg
};
P[80]{
   GP1:
	UF : 0, UT : 1,		CONFIG : 'N U T, 0, 0, 0',
	X = 1221.447  mm,	Y = -280.976  mm,	Z = -233.605  mm,
	W = 0.000 deg,	P = 30.000 deg,	R = -160.000 deg
};
P[81]{
   GP1:
	UF : 0, UT : 1,		CONFIG : 'N U T, 0, 0, 0',
	X = 1220.077  mm,	Y = -279.554  mm,	Z = -233.286  mm,
	W = 0.000 deg,	P = 30.000 deg,	R = -160.000 deg
};
P[82]{
   GP1:
	UF : 0, UT : 1,		CONFIG : 'N U T, 0, 0, 0',
	X = 1218.708  mm,	Y = -278.132  mm,	Z = -232.967  mm,
	W = 0.000 deg,	P = 30.000 deg,	R = -160.000 deg
};
P[83]{
   GP1:
	UF : 0, UT : 1,		CONFIG : 'N U T, 0, 0, 0',
	X = 1217.338  mm,	Y = -276.709  mm,	Z = -232.649  mm,
	W = 0.000 deg,	P = 30.000 deg,	R = -160.000 deg
};
P[84]{
   GP1:
	UF : 0, UT : 1,		CONFIG : 'N U T, 0, 0, 0',
	X = 1215.969  mm,	Y = -275.287  mm,	Z = -232.330  mm,
	W = 0.000 deg,	P = 30.000 deg,	R = -165.408 deg
};
P[85]{
   GP1:
	UF : 0, UT : 1,		CONFIG : 'N U T, 0, 0, 0',
	X = 1214.599  mm,	Y = -273.865  mm,	Z = -232.012  mm,
	W = 0.000 deg,	P = 30.000 deg,	R = -169.372 deg
};
P[86]{
   GP1:
	UF : 0, UT : 1,		CONFIG : 'N U T, 0, 0, 0',
	X = 1213.229  mm,	Y = -272.443  mm,	Z = -231.693  mm,
	W = 0.000 deg,	P = 30.000 deg,	R = -173.335 deg
};
P[87]{
   GP1:
	UF : 0, UT : 1,		CONFIG : 'N U T, 0, 0, 0',
	X = 1211.860  mm,	Y = -271.021  mm,	Z = -231.374  mm,
	W = 0.000 deg,	P = 30.000 deg,	R = -177.299 deg
};
P[88]{
   GP1:
	UF : 0, UT : 1,		CONFIG : 'N U T, 0, 0, 0',
	X = 1210.490  mm,	Y = -269.599  mm,	Z = -231.056  mm,
	W = 0.000 deg,	P = 30.000 deg,	R = -179.818 deg
};
P[89]{
   GP1:
	UF : 0, UT : 1,		CONFIG : 'N U T, 0, 0, 0',
	X = 1207.952  mm,	Y = -266.348  mm,	Z = -230.860  mm,
	W = 0.000 deg,	P = 30.000 deg,	R = -179.818 deg
};
P[90]{
   GP1:
	UF : 0, UT : 1,		CONFIG : 'N U T, 0, 0, 0',
	X = 1206.850  mm,	Y = -261.048  mm,	Z = -230.852  mm,
	W = 0.000 deg,	P = 30.000 deg,	R = -179.818 deg
};
P[91]{
   GP1:
	UF : 0, UT : 1,		CONFIG : 'N U T, 0, 0, 0',
	X = 1206.844  mm,	Y = -259.048  mm,	Z = -230.832  mm,
	W = 0.000 deg,	P = 30.000 deg,	R = -179.818 deg
};
P[92]{
   GP1:
	UF : 0, UT : 1,		CONFIG : 'N U T, 0, 0, 0',
	X = 1206.838  mm,	Y = -257.048  mm,	Z = -230.812  mm,
	W = 0.000 deg,	P = 30.000 deg,	R = -179.818 deg
};
P[93]{
   GP1:
	UF : 0, UT : 1,		CONFIG : 'N U T, 0, 0, 0',
	X = 1206.831  mm,	Y = -255.048  mm,	Z = -230.792  mm,
	W = 0.000 deg,	P = 30.000 deg,	R = -179.818 deg
};
P[94]{
   GP1:
	UF : 0, UT : 1,		CONFIG : 'N U T, 0, 0, 0',
	X = 1206.825  mm,	Y = -253.049  mm,	Z = -230.772  mm,
	W = 0.000 deg,	P = 30.000 deg,	R = -179.818 deg
};
P[95]{
   GP1:
	UF : 0, UT : 1,		CONFIG : 'N U T, 0, 0, 0',
	X = 1206.819  mm,	Y = -251.049  mm,	Z = -230.752  mm,
	W = 0.000 deg,	P = 30.000 deg,	R = -179.818 deg
};
P[96]{
   GP1:
	UF : 0, UT : 1,		CONFIG : 'N U T, 0, 0, 0',
	X = 1206.812  mm,	Y = -249.049  mm,	Z = -230.732  mm,
	W = 0.000 deg,	P = 30.000 deg,	R = -179.818 deg
};
P[97]{
   GP1:
	UF : 0, UT : 1,		CONFIG : 'N U T, 0, 0, 0',
	X = 1206.806  mm,	Y = -247.049  mm,	Z = -230.712  mm,
	W = 0.000 deg,	P = 30.000 deg,	R = -179.818 deg
};
P[98]{
   GP1:
	UF : 0, UT : 1,		CONFIG : 'N U T, 0, 0, 0',
	X = 1206.800  mm,	Y = -245.049  mm,	Z = -230.692  mm,
	W = 0.000 deg,	P = 30.000 deg,	R = -179.818 deg
};
P[99]{
   GP1:
	UF : 0, UT : 1,		CONFIG : 'N U T, 0, 0, 0',
	X = 1206.793  mm,	Y = -243.049  mm,	Z = -230.672  mm,
	W = 0.000 deg,	P = 30.000 deg,	R = -179.818 deg
};
P[100]{
   GP1:
	UF : 0, UT : 1,		CONFIG : 'N U T, 0, 0, 0',
	X = 1206.787  mm,	Y = -241.049  mm,	Z = -230.652  mm,
	W = 0.000 deg,	P = 30.000 deg,	R = -179.818 deg
};
P[101]{
   GP1:
	UF : 0, UT : 1,		CONFIG : 'N U T, 0, 0, 0',
	X = 1206.781  mm,	Y = -239.049  mm,	Z = -230.632  mm,
	W = 0.000 deg,	P = 30.000 deg,	R = -179.818 deg
};
P[102]{
   GP1:
	UF : 0, UT : 1,		CONFIG : 'N U T, 0, 0, 0',
	X = 1206.774  mm,	Y = -237.049  mm,	Z = -230.612  mm,
	W = 0.000 deg,	P = 30.000 deg,	R = -179.818 deg
};
P[103]{
   GP1:
	UF : 0, UT : 1,		CONFIG : 'N U T, 0, 0, 0',
	X = 1206.768  mm,	Y = -235.050  mm,	Z = -230.592  mm,
	W = 0.000 deg,	P = 30.000 deg,	R = -179.818 deg
};
P[104]{
   GP1:
	UF : 0, UT : 1,		CONFIG : 'N U T, 0, 0, 0',
	X = 1206.762  mm,	Y = -233.050  mm,	Z = -230.572  mm,
	W = 0.000 deg,	P = 30.000 deg,	R = -179.818 deg
};
P[105]{
   GP1:
	UF : 0, UT : 1,		CONFIG : 'N U T, 0, 0, 0',
	X = 1206.755  mm,	Y = -231.050  mm,	Z = -230.552  mm,
	W = 0.000 deg,	P = 30.000 deg,	R = -179.818 deg
};
P[106]{
   GP1:
	UF : 0, UT : 1,		CONFIG : 'N U T, 0, 0, 0',
	X = 1206.749  mm,	Y = -229.050  mm,	Z = -230.532  mm,
	W = 0.000 deg,	P = 30.000 deg,	R = -179.818 deg
};
P[107]{
   GP1:
	UF : 0, UT : 1,		CONFIG : 'N U T, 0, 0, 0',
	X = 1206.742  mm,	Y = -227.050  mm,	Z = -230.512  mm,
	W = 0.000 deg,	P = 30.000 deg,	R = -179.818 deg
};
P[108]{
   GP1:
	UF : 0, UT : 1,		CONFIG : 'N U T, 0, 0, 0',
	X = 1206.736  mm,	Y = -225.050  mm,	Z = -230.492  mm,
	W = 0.000 deg,	P = 30.000 deg,	R = -179.818 deg
};
P[109]{
   GP1:
	UF : 0, UT : 1,		CONFIG : 'N U T, 0, 0, 0',
	X = 1206.730  mm,	Y = -223.050  mm,	Z = -230.472  mm,
	W = 0.000 deg,	P = 30.000 deg,	R = -179.818 deg
};
P[110]{
   GP1:
	UF : 0, UT : 1,		CONFIG : 'N U T, 0, 0, 0',
	X = 1206.723  mm,	Y = -221.050  mm,	Z = -230.452  mm,
	W = 0.000 deg,	P = 30.000 deg,	R = -179.818 deg
};
P[111]{
   GP1:
	UF : 0, UT : 1,		CONFIG : 'N U T, 0, 0, 0',
	X = 1206.717  mm,	Y = -219.050  mm,	Z = -230.432  mm,
	W = 0.000 deg,	P = 30.000 deg,	R = -179.818 deg
};
P[112]{
   GP1:
	UF : 0, UT : 1,		CONFIG : 'N U T, 0, 0, 0',
	X = 1206.711  mm,	Y = -217.051  mm,	Z = -230.412  mm,
	W = 0.000 deg,	P = 30.000 deg,	R = -179.818 deg
};
P[113]{
   GP1:
	UF : 0, UT : 1,		CONFIG : 'N U T, 0, 0, 0',
	X = 1206.704  mm,	Y = -215.051  mm,	Z = -230.392  mm,
	W = 0.000 deg,	P = 30.000 deg,	R = -179.818 deg
};
P[114]{
   GP1:
	UF : 0, UT : 1,		CONFIG : 'N U T, 0, 0, 0',
	X = 1206.698  mm,	Y = -213.051  mm,	Z = -230.372  mm,
	W = 0.000 deg,	P = 30.000 deg,	R = -179.818 deg
};
P[115]{
   GP1:
	UF : 0, UT : 1,		CONFIG : 'N U T, 0, 0, 0',
	X = 1206.692  mm,	Y = -211.051  mm,	Z = -230.352  mm,
	W = 0.000 deg,	P = 30.000 deg,	R = -179.818 deg
};
P[116]{
   GP1:
	UF : 0, UT : 1,		CONFIG : 'N U T, 0, 0, 0',
	X = 1206.685  mm,	Y = -209.051  mm,	Z = -230.332  mm,
	W = 0.000 deg,	P = 30.000 deg,	R = 174.586 deg
};
P[117]{
   GP1:
	UF : 0, UT : 1,		CONFIG : 'N U T, 0, 0, 0',
	X = 1206.679  mm,	Y = -207.051  mm,	Z = -230.312  mm,
	W = 0.000 deg,	P = 30.000 deg,	R = 170.549 deg
};
P[118]{
   GP1:
	UF : 0, UT : 1,		CONFIG : 'N U T, 0, 0, 0',
	X = 1206.673  mm,	Y = -205.051  mm,	Z = -230.292  mm,
	W = 0.000 deg,	P = 30.000 deg,	R = 166.513 deg
};
P[119]{
   GP1:
	UF : 0, UT : 1,		CONFIG : 'N U T, 0, 0, 0',
	X = 1206.666  mm,	Y = -203.051  mm,	Z = -230.272  mm,
	W = 0.000 deg,	P = 30.000 deg,	R = 162.476 deg
};
P[120]{
   GP1:
	UF : 0, UT : 1,		CONFIG : 'N U T, 0, 0, 0',
	X = 1206.661  mm,	Y = -200.917  mm,	Z = -230.252  mm,
	W = 0.000 deg,	P = 30.000 deg,	R = 160.000 deg
};
P[121]{
   GP1:
	UF : 0, UT : 1,		CONFIG : 'N U T, 0, 0, 0',
	X = 1209.158  mm,	Y = -194.467  mm,	Z = -230.260  mm,
	W = 0.000 deg,	P = 30.000 deg,	R = 160.000 deg
};
P[122]{
   GP1:
	UF : 0, UT : 1,		CONFIG : 'N U T, 0, 0, 0',
	X = 1210.458  mm,	Y = -192.973  mm,	Z = -230.542  mm,
	W = 0.000 deg,	P = 30.000 deg,	R = 160.000 deg
};
P[123]{
   GP1:
	UF : 0, UT : 1,		CONFIG : 'N U T, 0, 0, 0',
	X = 1211.759  mm,	Y = -191.480  mm,	Z = -230.824  mm,
	W = 0.000 deg,	P = 30.000 deg,	R = 160.000 deg
};
P[124]{
   GP1:
	UF : 0, UT : 1,		CONFIG : 'N U T, 0, 0, 0',
	X = 1213.059  mm,	Y = -189.987  mm,	Z = -231.105  mm,
	W = 0.000 deg,	P = 30.000 deg,	R = 160.000 deg
};
P[125]{
   GP1:
	UF : 0, UT : 1,		CONFIG : 'N U T, 0, 0, 0',
	X = 1214.360  mm,	Y = -188.494  mm,	Z = -231.387  mm,
	W = 0.000 deg,	P = 30.000 deg,	R = 160.000 deg
};
P[126]{
   GP1:
	UF : 0, UT : 1,		CONFIG : 'N U T, 0, 0, 0',
	X = 1215.660  mm,	Y = -187.001  mm,	Z = -231.668  mm,
	W = 0.000 deg,	P = 30.000 deg,	R = 160.000 deg
};
P[127]{
   GP1:
	UF : 0, UT : 1,		CONFIG : 'N U T, 0, 0, 0',
	X = 1216.961  mm,	Y = -185.508  mm,	Z = -231.950  mm,
	W = 0.000 deg,	P = 30.000 deg,	R = 160.000 deg
};
P[128]{
   GP1:
	UF : 0, UT : 1,		CONFIG : 'N U T, 0, 0, 0',
	X = 1218.261  mm,	Y = -184.015  mm,	Z = -232.231  mm,
	W = 0.000 deg,	P = 30.000 deg,	R = 160.000 deg
};
P[129]{
   GP1:
	UF : 0, UT : 1,		CONFIG : 'N U T, 0, 0, 0',
	X = 1219.562  mm,	Y = -182.522  mm,	Z = -232.513  mm,
	W = 0.000 deg,	P = 30.000 deg,	R = 160.000 deg
};
P[130]{
   GP1:
	UF : 0, UT : 1,		CONFIG : 'N U T, 0, 0, 0',
	X = 1220.862  mm,	Y = -181.029  mm,	Z = -232.794  mm,
	W = 0.000 deg,	P = 30.000 deg,	R = 160.000 deg
};
P[131]{
   GP1:
	UF : 0, UT : 1,		CONFIG : 'N U T, 0, 0, 0',
	X = 1222.163  mm,	Y = -179.535  mm,	Z = -233.076  mm,
	W = 0.000 deg,	P = 30.000 deg,	R = 160.000 deg
};
P[132]{
   GP1:
	UF : 0, UT : 1,		CONFIG : 'N U T, 0, 0, 0',
	X = 1223.463  mm,	Y = -178.042  mm,	Z = -233.358  mm,
	W = 0.000 deg,	P = 30.000 deg,	R = 160.000 deg
};
P[133]{
   GP1:
	UF : 0, UT : 1,		CONFIG : 'N U T, 0, 0, 0',
	X = 1224.764  mm,	Y = -176.549  mm,	Z = -233.639  mm,
	W = 0.000 deg,	P = 30.000 deg,	R = 160.000 deg
};
P[134]{
   GP1:
	UF : 0, UT : 1,		CONFIG : 'N U T, 0, 0, 0',
	X = 1226.064  mm,	Y = -175.056  mm,	Z = -233.921  mm,
	W = 0.000 deg,	P = 30.000 deg,	R = 160.000 deg
};
P[135]{
   GP1:
	UF : 0, UT : 1,		CONFIG : 'N U T, 0, 0, 0',
	X = 1227.365  mm,	Y = -173.563  mm,	Z = -234.202  mm,
	W = 0.000 deg,	P = 30.000 deg,	R = 160.000 deg
};
P[136]{
   GP1:
	UF : 0, UT : 1,		CONFIG : 'N U T, 0, 0, 0',
	X = 1228.665  mm,	Y = -172.070  mm,	Z = -234.484  mm,
	W = 0.000 deg,	P = 30.000 deg,	R = 160.000 deg
};
P[137]{
   GP1:
	UF : 0, UT : 1,		CONFIG : 'N U T, 0, 0, 0',
	X = 1229.966  mm,	Y = -170.577  mm,	Z = -234.765  mm,
	W = 0.000 deg,	P = 30.000 deg,	R = 160.000 deg
};
P[138]{
   GP1:
	UF : 0, UT : 1,		CONFIG : 'N U T, 0, 0, 0',
	X = 1231.266  mm,	Y = -169.084  mm,	Z = -235.047  mm,
	W = 0.000 deg,	P = 30.000 deg,	R = 160.000 deg
};
P[139]{
   GP1:
	UF : 0, UT : 1,		CONFIG : 'N U T, 0, 0, 0',
	X = 1232.567  mm,	Y = -167.591  mm,	Z = -235.329  mm,
	W = 0.000 deg,	P = 30.000 deg,	R = 160.000 deg
};
P[140]{
   GP1:
	UF : 0, UT : 1,		CONFIG : 'N U T, 0, 0, 0',
	X = 1233.868  mm,	Y = -166.098  mm,	Z = -235.610  mm,
	W = 0.000 deg,	P = 30.000 deg,	R = 160.000 deg
};
P[141]{
   GP1:
	UF : 0, UT : 1,		CONFIG : 'N U T, 0, 0, 0',
	X = 1235.168  mm,	Y = -164.604  mm,	Z = -235.892  mm,
	W = 0.000 deg,	P = 30.000 deg,	R = 160.000 deg
};
P[142]{
   GP1:
	UF : 0, UT : 1,		CONFIG : 'N U T, 0, 0, 0',
	X = 1236.469  mm,	Y = -163.111  mm,	Z = -236.173  mm,
	W = 0.000 deg,	P = 30.000 deg,	R = 164.616 deg
};
P[143]{
   GP1:
	UF : 0, UT : 1,		CONFIG : 'N U T, 0, 0, 0',
	X = 1237.769  mm,	Y = -161.618  mm,	Z = -236.455  mm,
	W = 0.000 deg,	P = 30.000 deg,	R = 169.100 deg
};
P[144]{
   GP1:
	UF : 0, UT : 1,		CONFIG : 'N U T, 0, 0, 0',
	X = 1239.070  mm,	Y = -160.125  mm,	Z = -236.736  mm,
	W = 0.000 deg,	P = 30.000 deg,	R = 173.584 deg
};
P[145]{
   GP1:
	UF : 0, UT : 1,		CONFIG : 'N U T, 0, 0, 0',
	X = 1240.370  mm,	Y = -158.632  mm,	Z = -237.018  mm,
	W = 0.000 deg,	P = 30.000 deg,	R = 178.068 deg
};
P[146]{
   GP1:
	UF : 0, UT : 1,		CONFIG : 'N U T, 0, 0, 0',
	X = 1241.671  mm,	Y = -157.139  mm,	Z = -237.299  mm,
	W = 0.000 deg,	P = 30.000 deg,	R = -177.580 deg
};
P[147]{
   GP1:
	UF : 0, UT : 1,		CONFIG : 'N U T, 0, 0, 0',
	X = 1240.986  mm,	Y = -158.504  mm,	Z = -237.477  mm,
	W = 0.000 deg,	P = 30.000 deg,	R = -177.580 deg
};
P[148]{
   GP1:
	UF : 0, UT : 1,		CONFIG : 'N U T, 0, 0, 0',
	X = 1240.011  mm,	Y = -162.450  mm,	Z = -237.459  mm,
	W = 0.000 deg,	P = 30.000 deg,	R = -177.580 deg
};
P[149]{
   GP1:
	UF : 0, UT : 1,		CONFIG : 'N U T, 0, 0, 0',
	X = 1239.926  mm,	Y = -160.453  mm,	Z = -237.408  mm,
	W = 0.000 deg,	P = 30.000 deg,	R = -177.580 deg
};
P[150]{
   GP1:
	UF : 0, UT : 1,		CONFIG : 'N U T, 0, 0, 0',
	X = 1239.842  mm,	Y = -158.455  mm,	Z = -237.358  mm,
	W = 0.000 deg,	P = 30.000 deg,	R = -177.580 deg
};
P[151]{
   GP1:
	UF : 0, UT : 1,		CONFIG : 'N U T, 0, 0, 0',
	X = 1239.757  mm,	Y = -156.458  mm,	Z = -237.307  mm,
	W = 0.000 deg,	P = 30.000 deg,	R = -177.580 deg
};
P[152]{
   GP1:
	UF : 0, UT : 1,		CONFIG : 'N U T, 0, 0, 0',
	X = 1239.673  mm,	Y = -154.460  mm,	Z = -237.256  mm,
	W = 0.000 deg,	P = 30.000 deg,	R = -177.580 deg
};
P[153]{
   GP1:
	UF : 0, UT : 1,		CONFIG : 'N U T, 0, 0, 0',
	X = 1239.589  mm,	Y = -152.462  mm,	Z = -237.206  mm,
	W = 0.000 deg,	P = 30.000 deg,	R = -177.580 deg
};
P[154]{
   GP1:
	UF : 0, UT : 1,		CONFIG : 'N U T, 0, 0, 0',
	X = 1239.504  mm,	Y = -150.465  mm,	Z = -237.155  mm,
	W = 0.000 deg,	P = 30.000 deg,	R = -177.580 deg
};
P[155]{
   GP1:
	UF : 0, UT : 1,		CONFIG : 'N U T, 0, 0, 0',
	X = 1239.420  mm,	Y = -148.467  mm,	Z = -237.105  mm,
	W = 0.000 deg,	P = 30.000 deg,	R = -177.580 deg
};
P[156]{
   GP1:
	UF : 0, UT : 1,		CONFIG : 'N U T, 0, 0, 0',
	X = 1239.335  mm,	Y = -146.470  mm,	Z = -237.054  mm,
	W = 0.000 deg,	P = 30.000 deg,	R = -177.580 deg
};
P[157]{
   GP1:
	UF : 0, UT : 1,		CONFIG : 'N U T, 0, 0, 0',
	X = 1239.251  mm,	Y = -144.472  mm,	Z = -237.003  mm,
	W = 0.000 deg,	P = 30.000 deg,	R = -177.580 deg
};
P[158]{
   GP1:
	UF : 0, UT : 1,		CONFIG : 'N U T, 0, 0, 0',
	X = 1239.166  mm,	Y = -142.475  mm,	Z = -236.953  mm,
	W = 0.000 deg,	P = 30.000 deg,	R = -177.580 deg
};
P[159]{
   GP1:
	UF : 0, UT : 1,		CONFIG : 'N U T, 0, 0, 0',
	X = 1239.082  mm,	Y = -140.477  mm,	Z = -236.902  mm,
	W = 0.000 deg,	P = 30.000 deg,	R = -177.580 deg
};
P[160]{
   GP1:
	UF : 0, UT : 1,		CONFIG : 'N U T, 0, 0, 0',
	X = 1238.997  mm,	Y = -138.479  mm,	Z = -236.852  mm,
	W = 0.000 deg,	P = 30.000 deg,	R = -177.580 deg
};
P[161]{
   GP1:
	UF : 0, UT : 1,		CONFIG : 'N U T, 0, 0, 0',
	X = 1238.913  mm,	Y = -136.482  mm,	Z = -236.801  mm,
	W = 0.000 deg,	P = 30.000 deg,	R = -177.580 deg
};
P[162]{
   GP1:
	UF : 0, UT : 1,		CONFIG : 'N U T, 0, 0, 0',
	X = 1238.829  mm,	Y = -134.484  mm,	Z = -236.750  mm,
	W = 0.000 deg,	P = 30.000 deg,	R = -177.580 deg
};
P[163]{
   GP1:
	UF : 0, UT : 1,		CONFIG : 'N U T, 0, 0, 0',
	X = 1238.744  mm,	Y = -132.487  mm,	Z = -236.700  mm,
	W = 0.000 deg,	P = 30.000 deg,	R = -177.580 deg
};
P[164]{
   GP1:
	UF : 0, UT : 1,		CONFIG : 'N U T, 0, 0, 0',
	X = 1238.660  mm,	Y = -130.489  mm,	Z = -236.649  mm,
	W = 0.000 deg,	P = 30.000 deg,	R = -177.580 deg
};
P[165]{
   GP1:
	UF : 0, UT : 1,		CONFIG : 'N U T, 0, 0, 0',
	X = 1238.575  mm,	Y = -128.492  mm,	Z = -236.599  mm,
	W = 0.000 deg,	P = 30.000 deg,	R = -177.580 deg
};
P[166]{
   GP1:
	UF : 0, UT : 1,		CONFIG : 'N U T, 0, 0, 0',
	X = 1238.491  mm,	Y = -126.494  mm,	Z = -236.548  mm,
	W = 0.000 deg,	P = 30.000 deg,	R = -177.580 deg
};
P[167]{
   GP1:
	UF : 0, UT : 1,		CONFIG : 'N U T, 0, 0, 0',
	X = 1238.406  mm,	Y = -124.496  mm,	Z = -236.497  mm,
	W = 0.000 deg,	P = 30.000 deg,	R = -177.580 deg
};
P[168]{
   GP1:
	UF : 0, UT : 1,		CONFIG : 'N U T, 0, 0, 0',
	X = 1238.322  mm,	Y = -122.499  mm,	Z = -236.447  mm,
	W = 0.000 deg,	P = 30.000 deg,	R = -177.580 deg
};
P[169]{
   GP1:
	UF : 0, UT : 1,		CONFIG : 'N U T, 0, 0, 0',
	X = 1238.238  mm,	Y = -120.501  mm,	Z = -236.396  mm,
	W = 0.000 deg,	P = 30.000 deg,	R = -177.580 deg
};
P[170]{
   GP1:
	UF : 0, UT : 1,		CONFIG : 'N U T, 0, 0, 0',
	X = 1238.153  mm,	Y = -118.504  mm,	Z = -236.346  mm,
	W = 0.000 deg,	P = 30.000 deg,	R = -177.580 deg
};
P[171]{
   GP1:
	UF : 0, UT : 1,		CONFIG : 'N U T, 0, 0, 0',
	X = 1238.069  mm,	Y = -116.506  mm,	Z = -236.295  mm,
	W = 0.000 deg,	P = 30.000 deg,	R = -177.580 deg
};
P[172]{
   GP1:
	UF : 0, UT : 1,		CONFIG : 'N U T, 0, 0, 0',
	X = 1237.984  mm,	Y = -114.509  mm,	Z = -236.244  mm,
	W = 0.000 deg,	P = 30.000 deg,	R = -172.769 deg
};
P[173]{
   GP1:
	UF : 0, UT : 1,		CONFIG : 'N U T, 0, 0, 0',
	X = 1237.900  mm,	Y = -112.511  mm,	Z = -236.194  mm,
	W = 0.000 deg,	P = 30.000 deg,	R = -169.253 deg
};
P[174]{
   GP1:
	UF : 0, UT : 1,		CONFIG : 'N U T, 0, 0, 0',
	X = 1237.815  mm,	Y = -110.513  mm,	Z = -236.143  mm,
	W = 0.000 deg,	P = 30.000 deg,	R = -165.737 deg
};
P[175]{
   GP1:
	UF : 0, UT : 1,		CONFIG : 'N U T, 0, 0, 0',
	X = 1237.731  mm,	Y = -108.516  mm,	Z = -236.093  mm,
	W = 0.000 deg,	P = 30.000 deg,	R = -162.221 deg
};
P[176]{
   GP1:
	UF : 0, UT : 1,		CONFIG : 'N U T, 0, 0, 0',
	X = 1237.646  mm,	Y = -106.518  mm,	Z = -236.042  mm,
	W = 0.000 deg,	P = 30.000 deg,	R = -160.000 deg
};
P[177]{
   GP1:
	UF : 0, UT : 1,		CONFIG : 'N U T, 0, 0, 0',
	X = 1240.484  mm,	Y = -113.055  mm,	Z = -236.041  mm,
	W = 0.000 deg,	P = 30.000 deg,	R = -160.000 deg
};
P[178]{
   GP1:
	UF : 0, UT : 1,		CONFIG : 'N U T, 0, 0, 0',
	X = 1239.184  mm,	Y = -111.752  mm,	Z = -235.722  mm,
	W = 0.000 deg,	P = 30.000 deg,	R = -160.000 deg
};
P[179]{
   GP1:
	UF : 0, UT : 1,		CONFIG : 'N U T, 0, 0, 0',
	X = 1237.790  mm,	Y = -110.355  mm,	Z = -235.397  mm,
	W = 0.000 deg,	P = 30.000 deg,	R = -160.000 deg
};
P[180]{
   GP1:
	UF : 0, UT : 1,		CONFIG : 'N U T, 0, 0, 0',
	X = 1236.396  mm,	Y = -108.958  mm,	Z = -235.072  mm,
	W = 0.000 deg,	P = 30.000 deg,	R = -160.000 deg
};
P[181]{
   GP1:
	UF : 0, UT : 1,		CONFIG : 'N U T, 0, 0, 0',
	X = 1235.003  mm,	Y = -107.561  mm,	Z = -234.748  mm,
	W = 0.000 deg,	P = 30.000 deg,	R = -160.000 deg
};
P[182]{
   GP1:
	UF : 0, UT : 1,		CONFIG : 'N U T, 0, 0, 0',
	X = 1233.609  mm,	Y = -106.164  mm,	Z = -234.423  mm,
	W = 0.000 deg,	P = 30.000 deg,	R = -160.000 deg
};
P[183]{
   GP1:
	UF : 0, UT : 1,		CONFIG : 'N U T, 0, 0, 0',
	X = 1232.215  mm,	Y = -104.767  mm,	Z = -234.099  mm,
	W = 0.000 deg,	P = 30.000 deg,	R = -160.000 deg
};
P[184]{
   GP1:
	UF : 0, UT : 1,		CONFIG : 'N U T, 0, 0, 0',
	X = 1230.821  mm,	Y = -103.370  mm,	Z = -233.774  mm,
	W = 0.000 deg,	P = 30.000 deg,	R = -160.000 deg
};
P[185]{
   GP1:
	UF : 0, UT : 1,		CONFIG : 'N U T, 0, 0, 0',
	X = 1229.427  mm,	Y = -101.973  mm,	Z = -233.449  mm,
	W = 0.000 deg,	P = 30.000 deg,	R = -160.000 deg
};
P[186]{
   GP1:
	UF : 0, UT : 1,		CONFIG : 'N U T, 0, 0, 0',
	X = 1228.034  mm,	Y = -100.575  mm,	Z = -233.125  mm,
	W = 0.000 deg,	P = 30.000 deg,	R = -160.000 deg
};
P[187]{
   GP1:
	UF : 0, UT : 1,		CONFIG : 'N U T, 0, 0, 0',
	X = 1226.640  mm,	Y = -99.178  mm,	Z = -232.800  mm,
	W = 0.000 deg,	P = 30.000 deg,	R = -160.000 deg
};
P[188]{
   GP1:
	UF : 0, UT : 1,		CONFIG : 'N U T, 0, 0, 0',
	X = 1225.246  mm,	Y = -97.781  mm,	Z = -232.476  mm,
	W = 0.000 deg,	P = 30.000 deg,	R = -160.000 deg
};
P[189]{
   GP1:
	UF : 0, UT : 1,		CONFIG : 'N U T, 0, 0, 0',
	X = 1223.852  mm,	Y = -96.384  mm,	Z = -232.151  mm,
	W = 0.000 deg,	P = 30.000 deg,	R = -160.000 deg
};
P[190]{
   GP1:
	UF : 0, UT : 1,		CONFIG : 'N U T, 0, 0, 0',
	X = 1222.458  mm,	Y = -94.987  mm,	Z = -231.827  mm,
	W = 0.000 deg,	P = 30.000 deg,	R = -160.000 deg
};
P[191]{
   GP1:
	UF : 0, UT : 1,		CONFIG : 'N U T, 0, 0, 0',
	X = 1221.065  mm,	Y = -93.590  mm,	Z = -231.502  mm,
	W = 0.000 deg,	P = 30.000 deg,	R = -160.000 deg
};
P[192]{
   GP1:
	UF : 0, UT : 1,		CONFIG : 'N U T, 0, 0, 0',
	X = 1219.671  mm,	Y = -92.193  mm,	Z = -231.177  mm,
	W = 0.000 deg,	P = 30.000 deg,	R = -160.000 deg
};
P[193]{
   GP1:
	UF : 0, UT : 1,		CONFIG : 'N U T, 0, 0, 0',
	X = 1218.277  mm,	Y = -90.796  mm,	Z = -230.853  mm,
	W = 0.000 deg,	P = 30.000 deg,	R = -160.000 deg
};
P[194]{
   GP1:
	UF : 0, UT : 1,		CONFIG : 'N U T, 0, 0, 0',
	X = 1216.883  mm,	Y = -89.399  mm,	Z = -230.528  mm,
	W = 0.000 deg,	P = 30.000 deg,	R = -160.000 deg
};
P[195]{
   GP1:
	UF : 0, UT : 1,		CONFIG : 'N U T, 0, 0, 0',
	X = 1215.489  mm,	Y = -88.001  mm,	Z = -230.204  mm,
	W = 0.000 deg,	P = 30.000 deg,	R = -160.000 deg
};
P[196]{
   GP1:
	UF : 0, UT : 1,		CONFIG : 'N U T, 0, 0, 0',
	X = 1214.095  mm,	Y = -86.604  mm,	Z = -229.879  mm,
	W = 0.000 deg,	P = 30.000 deg,	R = -160.000 deg
};
P[197]{
   GP1:
	UF : 0, UT : 1,		CONFIG : 'N U T, 0, 0, 0',
	X = 1212.702  mm,	Y = -85.207  mm,	Z = -229.554  mm,
	W = 0.000 deg,	P = 30.000 deg,	R = -160.000 deg
};
P[198]{
   GP1:
	UF : 0, UT : 1,		CONFIG : 'N U T, 0, 0, 0',
	X = 1211.308  mm,	Y = -83.810  mm,	Z = -229.230  mm,
	W = 0.000 deg,	P = 30.000 deg,	R = -164.013 deg
};
P[199]{
   GP1:
	UF : 0, UT : 1,		CONFIG : 'N U T, 0, 0, 0',
	X = 1209.914  mm,	Y = -82.413  mm,	Z = -228.905  mm,
	W = 0.000 deg,	P = 30.000 deg,	R = -168.087 deg
};
P[200]{
   GP1:
	UF : 0, UT : 1,		CONFIG : 'N U T, 0, 0, 0',
	X = 1208.520  mm,	Y = -81.016  mm,	Z = -228.581  mm,
	W = 0.000 deg,	P = 30.000 deg,	R = -172.161 deg
};
P[201]{
   GP1:
	UF : 0, UT : 1,		CONFIG : 'N U T, 0, 0, 0',
	X = 1207.126  mm,	Y = -79.619  mm,	Z = -228.256  mm,
	W = 0.000 deg,	P = 30.000 deg,	R = -176.236 deg
};
P[202]{
   GP1:
	UF : 0, UT : 1,		CONFIG : 'N U T, 0, 0, 0',
	X = 1205.733  mm,	Y = -78.222  mm,	Z = -227.931  mm,
	W = 0.000 deg,	P = 30.000 deg,	R = 179.690 deg
};
P[203]{
   GP1:
	UF : 0, UT : 1,		CONFIG : 'N U T, 0, 0, 0',
	X = 1203.181  mm,	Y = -75.137  mm,	Z = -227.721  mm,
	W = 0.000 deg,	P = 30.000 deg,	R = 179.629 deg
};
P[204]{
   GP1:
	UF : 0, UT : 1,		CONFIG : 'N U T, 0, 0, 0',
	X = 1201.912  mm,	Y = -69.486  mm,	Z = -227.715  mm,
	W = 0.000 deg,	P = 30.000 deg,	R = 179.629 deg
};
P[205]{
   GP1:
	UF : 0, UT : 1,		CONFIG : 'N U T, 0, 0, 0',
	X = 1201.925  mm,	Y = -67.486  mm,	Z = -227.699  mm,
	W = 0.000 deg,	P = 30.000 deg,	R = 179.629 deg
};
P[206]{
   GP1:
	UF : 0, UT : 1,		CONFIG : 'N U T, 0, 0, 0',
	X = 1201.938  mm,	Y = -65.486  mm,	Z = -227.683  mm,
	W = 0.000 deg,	P = 30.000 deg,	R = 179.629 deg
};
P[207]{
   GP1:
	UF : 0, UT : 1,		CONFIG : 'N U T, 0, 0, 0',
	X = 1201.951  mm,	Y = -63.486  mm,	Z = -227.668  mm,
	W = 0.000 deg,	P = 30.000 deg,	R = 179.629 deg
};
P[208]{
   GP1:
	UF : 0, UT : 1,		CONFIG : 'N U T, 0, 0, 0',
	X = 1201.964  mm,	Y = -61.486  mm,	Z = -227.652  mm,
	W = 0.000 deg,	P = 30.000 deg,	R = 179.629 deg
};
P[209]{
   GP1:
	UF : 0, UT : 1,		CONFIG : 'N U T, 0, 0, 0',
	X = 1201.977  mm,	Y = -59.486  mm,	Z = -227.636  mm,
	W = 0.000 deg,	P = 30.000 deg,	R = 179.629 deg
};
P[210]{
   GP1:
	UF : 0, UT : 1,		CONFIG : 'N U T, 0, 0, 0',
	X = 1201.990  mm,	Y = -57.486  mm,	Z = -227.620  mm,
	W = 0.000 deg,	P = 30.000 deg,	R = 179.629 deg
};
P[211]{
   GP1:
	UF : 0, UT : 1,		CONFIG : 'N U T, 0, 0, 0',
	X = 1202.003  mm,	Y = -55.486  mm,	Z = -227.604  mm,
	W = 0.000 deg,	P = 30.000 deg,	R = 179.629 deg
};
P[212]{
   GP1:
	UF : 0, UT : 1,		CONFIG : 'N U T, 0, 0, 0',
	X = 1202.016  mm,	Y = -53.486  mm,	Z = -227.588  mm,
	W = 0.000 deg,	P = 30.000 deg,	R = 179.629 deg
};
P[213]{
   GP1:
	UF : 0, UT : 1,		CONFIG : 'N U T, 0, 0, 0',
	X = 1202.028  mm,	Y = -51.487  mm,	Z = -227.573  mm,
	W = 0.000 deg,	P = 30.000 deg,	R = 179.629 deg
};
P[214]{
   GP1:
	UF : 0, UT : 1,		CONFIG : 'N U T, 0, 0, 0',
	X = 1202.041  mm,	Y = -49.487  mm,	Z = -227.557  mm,
	W = 0.000 deg,	P = 30.000 deg,	R = 179.629 deg
};
P[215]{
   GP1:
	UF : 0, UT : 1,		CONFIG : 'N U T, 0, 0, 0',
	X = 1202.054  mm,	Y = -47.487  mm,	Z = -227.541  mm,
	W = 0.000 deg,	P = 30.000 deg,	R = 179.629 deg
};
P[216]{
   GP1:
	UF : 0, UT : 1,		CONFIG : 'N U T, 0, 0, 0',
	X = 1202.067  mm,	Y = -45.487  mm,	Z = -227.525  mm,
	W = 0.000 deg,	P = 30.000 deg,	R = 179.629 deg
};
P[217]{
   GP1:
	UF : 0, UT : 1,		CONFIG : 'N U T, 0, 0, 0',
	X = 1202.080  mm,	Y = -43.487  mm,	Z = -227.509  mm,
	W = 0.000 deg,	P = 30.000 deg,	R = 179.629 deg
};
P[218]{
   GP1:
	UF : 0, UT : 1,		CONFIG : 'N U T, 0, 0, 0',
	X = 1202.093  mm,	Y = -41.487  mm,	Z = -227.494  mm,
	W = 0.000 deg,	P = 30.000 deg,	R = 179.629 deg
};
P[219]{
   GP1:
	UF : 0, UT : 1,		CONFIG : 'N U T, 0, 0, 0',
	X = 1202.106  mm,	Y = -39.487  mm,	Z = -227.478  mm,
	W = 0.000 deg,	P = 30.000 deg,	R = 179.629 deg
};
P[220]{
   GP1:
	UF : 0, UT : 1,		CONFIG : 'N U T, 0, 0, 0',
	X = 1202.119  mm,	Y = -37.487  mm,	Z = -227.462  mm,
	W = 0.000 deg,	P = 30.000 deg,	R = 179.629 deg
};
P[221]{
   GP1:
	UF : 0, UT : 1,		CONFIG : 'N U T, 0, 0, 0',
	X = 1202.132  mm,	Y = -35.487  mm,	Z = -227.446  mm,
	W = 0.000 deg,	P = 30.000 deg,	R = 179.629 deg
};
P[222]{
   GP1:
	UF : 0, UT : 1,		CONFIG : 'N U T, 0, 0, 0',
	X = 1202.145  mm,	Y = -33.487  mm,	Z = -227.430  mm,
	W = 0.000 deg,	P = 30.000 deg,	R = 179.629 deg
};
P[223]{
   GP1:
	UF : 0, UT : 1,		CONFIG : 'N U T, 0, 0, 0',
	X = 1202.158  mm,	Y = -31.488  mm,	Z = -227.414  mm,
	W = 0.000 deg,	P = 30.000 deg,	R = 179.629 deg
};
P[224]{
   GP1:
	UF : 0, UT : 1,		CONFIG : 'N U T, 0, 0, 0',
	X = 1202.171  mm,	Y = -29.488  mm,	Z = -227.399  mm,
	W = 0.000 deg,	P = 30.000 deg,	R = 179.629 deg
};
P[225]{
   GP1:
	UF : 0, UT : 1,		CONFIG : 'N U T, 0, 0, 0',
	X = 1202.184  mm,	Y = -27.488  mm,	Z = -227.383  mm,
	W = 0.000 deg,	P = 30.000 deg,	R = 179.629 deg
};
P[226]{
   GP1:
	UF : 0, UT : 1,		CONFIG : 'N U T, 0, 0, 0',
	X = 1202.197  mm,	Y = -25.488  mm,	Z = -227.367  mm,
	W = 0.000 deg,	P = 30.000 deg,	R = 179.629 deg
};
P[227]{
   GP1:
	UF : 0, UT : 1,		CONFIG : 'N U T, 0, 0, 0',
	X = 1202.210  mm,	Y = -23.488  mm,	Z = -227.351  mm,
	W = 0.000 deg,	P = 30.000 deg,	R = 179.629 deg
};
P[228]{
   GP1:
	UF : 0, UT : 1,		CONFIG : 'N U T, 0, 0, 0',
	X = 1202.223  mm,	Y = -21.488  mm,	Z = -227.335  mm,
	W = 0.000 deg,	P = 30.000 deg,	R = 178.252 deg
};
P[229]{
   GP1:
	UF : 0, UT : 1,		CONFIG : 'N U T, 0, 0, 0',
	X = 1202.236  mm,	Y = -19.488  mm,	Z = -227.320  mm,
	W = 0.000 deg,	P = 30.000 deg,	R = 174.326 deg
};
P[230]{
   GP1:
	UF : 0, UT : 1,		CONFIG : 'N U T, 0, 0, 0',
	X = 1202.249  mm,	Y = -17.488  mm,	Z = -227.304  mm,
	W = 0.000 deg,	P = 30.000 deg,	R = 170.400 deg
};
P[231]{
   GP1:
	UF : 0, UT : 1,		CONFIG : 'N U T, 0, 0, 0',
	X = 1202.262  mm,	Y = -15.488  mm,	Z = -227.288  mm,
	W = 0.000 deg,	P = 30.000 deg,	R = 166.475 deg
};
P[232]{
   GP1:
	UF : 0, UT : 1,		CONFIG : 'N U T, 0, 0, 0',
	X = 1202.275  mm,	Y = -13.489  mm,	Z = -227.272  mm,
	W = 0.000 deg,	P = 30.000 deg,	R = 162.549 deg
};
P[233]{
   GP1:
	UF : 0, UT : 1,		CONFIG : 'N U T, 0, 0, 0',
	X = 1202.288  mm,	Y = -11.489  mm,	Z = -227.256  mm,
	W = 0.000 deg,	P = 30.000 deg,	R = 160.000 deg
};
P[234]{
   GP1:
	UF : 0, UT : 1,		CONFIG : 'N U T, 0, 0, 0',
	X = 1204.908  mm,	Y = -4.792  mm,	Z = -227.256  mm,
	W = 0.000 deg,	P = 30.000 deg,	R = 160.000 deg
};
P[235]{
   GP1:
	UF : 0, UT : 1,		CONFIG : 'N U T, 0, 0, 0',
	X = 1206.270  mm,	Y = -3.315  mm,	Z = -227.555  mm,
	W = 0.000 deg,	P = 30.000 deg,	R = 160.000 deg
};
P[236]{
   GP1:
	UF : 0, UT : 1,		CONFIG : 'N U T, 0, 0, 0',
	X = 1207.611  mm,	Y = -1.862  mm,	Z = -227.855  mm,
	W = 0.000 deg,	P = 30.000 deg,	R = 160.000 deg
};
P[237]{
   GP1:
	UF : 0, UT : 1,		CONFIG : 'N U T, 0, 0, 0',
	X = 1208.952  mm,	Y = -0.409  mm,	Z = -228.156  mm,
	W = 0.000 deg,	P = 30.000 deg,	R = 160.000 deg
};
P[238]{
   GP1:
	UF : 0, UT : 1,		CONFIG : 'N U T, 0, 0, 0',
	X = 1210.293  mm,	Y = 1.044  mm,	Z = -228.456  mm,
	W = 0.000 deg,	P = 30.000 deg,	R = 160.000 deg
};
P[239]{
   GP1:
	UF : 0, UT : 1,		CONFIG : 'N U T, 0, 0, 0',
	X = 1211.634  mm,	Y = 2.497  mm,	Z = -228.757  mm,
	W = 0.000 deg,	P = 30.000 deg,	R = 160.000 deg
};
P[240]{
   GP1:
	UF : 0, UT : 1,		CONFIG : 'N U T, 0, 0, 0',
	X = 1212.974  mm,	Y = 3.951  mm,	Z = -229.057  mm,
	W = 0.000 deg,	P = 30.000 deg,	R = 160.000 deg
};
P[241]{
   GP1:
	UF : 0, UT : 1,		CONFIG : 'N U T, 0, 0, 0',
	X = 1214.315  mm,	Y = 5.404  mm,	Z = -229.358  mm,
	W = 0.000 deg,	P = 30.000 deg,	R = 160.000 deg
};
P[242]{
   GP1:
	UF : 0, UT : 1,		CONFIG : 'N U T, 0, 0, 0',
	X = 1215.656  mm,	Y = 6.857  mm,	Z = -229.658  mm,
	W = 0.000 deg,	P = 30.000 deg,	R = 160.000 deg
};
P[243]{
   GP1:
	UF : 0, UT : 1,		CONFIG : 'N U T, 0, 0, 0',
	X = 1216.997  mm,	Y = 8.310  mm,	Z = -229.959  mm,
	W = 0.000 deg,	P = 30.000 deg,	R = 160.000 deg
};
P[244]{
   GP1:
	UF : 0, UT : 1,		CONFIG : 'N U T, 0, 0, 0',
	X = 1218.338  mm,	Y = 9.763  mm,	Z = -230.259  mm,
	W = 0.000 deg,	P = 30.000 deg,	R = 160.000 deg
};
P[245]{
   GP1:
	UF : 0, UT : 1,		CONFIG : 'N U T, 0, 0, 0',
	X = 1219.679  mm,	Y = 11.217  mm,	Z = -230.560  mm,
	W = 0.000 deg,	P = 30.000 deg,	R = 160.000 deg
};
P[246]{
   GP1:
	UF : 0, UT : 1,		CONFIG : 'N U T, 0, 0, 0',
	X = 1221.020  mm,	Y = 12.670  mm,	Z = -230.860  mm,
	W = 0.000 deg,	P = 30.000 deg,	R = 160.000 deg
};
P[247]{
   GP1:
	UF : 0, UT : 1,		CONFIG : 'N U T, 0, 0, 0',
	X = 1222.360  mm,	Y = 14.123  mm,	Z = -231.161  mm,
	W = 0.000 deg,	P = 30.000 deg,	R = 160.000 deg
};
P[248]{
   GP1:
	UF : 0, UT : 1,		CONFIG : 'N U T, 0, 0, 0',
	X = 1223.701  mm,	Y = 15.576  mm,	Z = -231.461  mm,
	W = 0.000 deg,	P = 30.000 deg,	R = 160.000 deg
};
P[249]{
   GP1:
	UF : 0, UT : 1,		CONFIG : 'N U T, 0, 0, 0',
	X = 1225.042  mm,	Y = 17.029  mm,	Z = -231.762  mm,
	W = 0.000 deg,	P = 30.000 deg,	R = 160.000 deg
};
P[250]{
   GP1:
	UF : 0, UT : 1,		CONFIG : 'N U T, 0, 0, 0',
	X = 1226.383  mm,	Y = 18.483  mm,	Z = -232.062  mm,
	W = 0.000 deg,	P = 30.000 deg,	R = 160.000 deg
};
P[251]{
   GP1:
	UF : 0, UT : 1,		CONFIG : 'N U T, 0, 0, 0',
	X = 1227.724  mm,	Y = 19.936  mm,	Z = -232.363  mm,
	W = 0.000 deg,	P = 30.000 deg,	R = 160.000 deg
};
P[252]{
   GP1:
	UF : 0, UT : 1,		CONFIG : 'N U T, 0, 0, 0',
	X = 1229.065  mm,	Y = 21.389  mm,	Z = -232.663  mm,
	W = 0.000 deg,	P = 30.000 deg,	R = 160.000 deg
};
P[253]{
   GP1:
	UF : 0, UT : 1,		CONFIG : 'N U T, 0, 0, 0',
	X = 1230.406  mm,	Y = 22.842  mm,	Z = -232.964  mm,
	W = 0.000 deg,	P = 30.000 deg,	R = 160.000 deg
};
P[254]{
   GP1:
	UF : 0, UT : 1,		CONFIG : 'N U T, 0, 0, 0',
	X = 1231.746  mm,	Y = 24.296  mm,	Z = -233.264  mm,
	W = 0.000 deg,	P = 30.000 deg,	R = 160.000 deg
};
P[255]{
   GP1:
	UF : 0, UT : 1,		CONFIG : 'N U T, 0, 0, 0',
	X = 1233.087  mm,	Y = 25.749  mm,	Z = -233.565  mm,
	W = 0.000 deg,	P = 30.000 deg,	R = 160.000 deg
};
P[256]{
   GP1:
	UF : 0, UT : 1,		CONFIG : 'N U T, 0, 0, 0',
	X = 1234.428  mm,	Y = 27.202  mm,	Z = -233.865  mm,
	W = 0.000 deg,	P = 30.000 deg,	R = 168.845 deg
};
P[257]{
   GP1:
	UF : 0, UT : 1,		CONFIG : 'N U T, 0, 0, 0',
	X = 1235.769  mm,	Y = 28.655  mm,	Z = -234.166  mm,
	W = 0.000 deg,	P = 30.000 deg,	R = 173.281 deg
};
P[258]{
   GP1:
	UF : 0, UT : 1,		CONFIG : 'N U T, 0, 0, 0',
	X = 1237.110  mm,	Y = 30.108  mm,	Z = -234.466  mm,
	W = 0.000 deg,	P = 30.000 deg,	R = 177.718 deg
};
P[259]{
   GP1:
	UF : 0, UT : 1,		CONFIG : 'N U T, 0, 0, 0',
	X = 1238.451  mm,	Y = 31.562  mm,	Z = -234.767  mm,
	W = 0.000 deg,	P = 30.000 deg,	R = -177.845 deg
};
P[260]{
   GP1:
	UF : 0, UT : 1,		CONFIG : 'N U T, 0, 0, 0',
	X = 1236.643  mm,	Y = 27.876  mm,	Z = -234.883  mm,
	W = 0.000 deg,	P = 30.000 deg,	R = -177.816 deg
};
P[261]{
   GP1:
	UF : 0, UT : 1,		CONFIG : 'N U T, 0, 0, 0',
	X = 1236.276  mm,	Y = 26.188  mm,	Z = -234.862  mm,
	W = 0.000 deg,	P = 30.000 deg,	R = -177.816 deg
};
P[262]{
   GP1:
	UF : 0, UT : 1,		CONFIG : 'N U T, 0, 0, 0',
	X = 1236.200  mm,	Y = 28.186  mm,	Z = -234.829  mm,
	W = 0.000 deg,	P = 30.000 deg,	R = -177.816 deg
};
P[263]{
   GP1:
	UF : 0, UT : 1,		CONFIG : 'N U T, 0, 0, 0',
	X = 1236.124  mm,	Y = 30.184  mm,	Z = -234.797  mm,
	W = 0.000 deg,	P = 30.000 deg,	R = -177.816 deg
};
P[264]{
   GP1:
	UF : 0, UT : 1,		CONFIG : 'N U T, 0, 0, 0',
	X = 1236.048  mm,	Y = 32.183  mm,	Z = -234.764  mm,
	W = 0.000 deg,	P = 30.000 deg,	R = -177.816 deg
};
P[265]{
   GP1:
	UF : 0, UT : 1,		CONFIG : 'N U T, 0, 0, 0',
	X = 1235.972  mm,	Y = 34.181  mm,	Z = -234.731  mm,
	W = 0.000 deg,	P = 30.000 deg,	R = -177.816 deg
};
P[266]{
   GP1:
	UF : 0, UT : 1,		CONFIG : 'N U T, 0, 0, 0',
	X = 1235.895  mm,	Y = 36.179  mm,	Z = -234.698  mm,
	W = 0.000 deg,	P = 30.000 deg,	R = -177.816 deg
};
P[267]{
   GP1:
	UF : 0, UT : 1,		CONFIG : 'N U T, 0, 0, 0',
	X = 1235.819  mm,	Y = 38.178  mm,	Z = -234.665  mm,
	W = 0.000 deg,	P = 30.000 deg,	R = -177.816 deg
};
P[268]{
   GP1:
	UF : 0, UT : 1,		CONFIG : 'N U T, 0, 0, 0',
	X = 1235.743  mm,	Y = 40.176  mm,	Z = -234.632  mm,
	W = 0.000 deg,	P = 30.000 deg,	R = -177.816 deg
};
P[269]{
   GP1:
	UF : 0, UT : 1,		CONFIG : 'N U T, 0, 0, 0',
	X = 1235.667  mm,	Y = 42.174  mm,	Z = -234.599  mm,
	W = 0.000 deg,	P = 30.000 deg,	R = -177.816 deg
};
P[270]{
   GP1:
	UF : 0, UT : 1,		CONFIG : 'N U T, 0, 0, 0',
	X = 1235.591  mm,	Y = 44.172  mm,	Z = -234.566  mm,
	W = 0.000 deg,	P = 30.000 deg,	R = -177.816 deg
};
P[271]{
   GP1:
	UF : 0, UT : 1,		CONFIG : 'N U T, 0, 0, 0',
	X = 1235.514  mm,	Y = 46.171  mm,	Z = -234.533  mm,
	W = 0.000 deg,	P = 30.000 deg,	R = -177.816 deg
};
P[272]{
   GP1:
	UF : 0, UT : 1,		CONFIG : 'N U T, 0, 0, 0',
	X = 1235.438  mm,	Y = 48.169  mm,	Z = -234.501  mm,
	W = 0.000 deg,	P = 30.000 deg,	R = -177.816 deg
};
P[273]{
   GP1:
	UF : 0, UT : 1,		CONFIG : 'N U T, 0, 0, 0',
	X = 1235.362  mm,	Y = 50.167  mm,	Z = -234.468  mm,
	W = 0.000 deg,	P = 30.000 deg,	R = -177.816 deg
};
P[274]{
   GP1:
	UF : 0, UT : 1,		CONFIG : 'N U T, 0, 0, 0',
	X = 1235.286  mm,	Y = 52.165  mm,	Z = -234.435  mm,
	W = 0.000 deg,	P = 30.000 deg,	R = -177.816 deg
};
P[275]{
   GP1:
	UF : 0, UT : 1,		CONFIG : 'N U T, 0, 0, 0',
	X = 1235.210  mm,	Y = 54.164  mm,	Z = -234.402  mm,
	W = 0.000 deg,	P = 30.000 deg,	R = -177.816 deg
};
P[276]{
   GP1:
	UF : 0, UT : 1,		CONFIG : 'N U T, 0, 0, 0',
	X = 1235.133  mm,	Y = 56.162  mm,	Z = -234.369  mm,
	W = 0.000 deg,	P = 30.000 deg,	R = -177.816 deg
};
P[277]{
   GP1:
	UF : 0, UT : 1,		CONFIG : 'N U T, 0, 0, 0',
	X = 1235.057  mm,	Y = 58.160  mm,	Z = -234.336  mm,
	W = 0.000 deg,	P = 30.000 deg,	R = -177.816 deg
};
P[278]{
   GP1:
	UF : 0, UT : 1,		CONFIG : 'N U T, 0, 0, 0',
	X = 1234.981  mm,	Y = 60.159  mm,	Z = -234.303  mm,
	W = 0.000 deg,	P = 30.000 deg,	R = -177.816 deg
};
P[279]{
   GP1:
	UF : 0, UT : 1,		CONFIG : 'N U T, 0, 0, 0',
	X = 1234.905  mm,	Y = 62.157  mm,	Z = -234.270  mm,
	W = 0.000 deg,	P = 30.000 deg,	R = -177.816 deg
};
P[280]{
   GP1:
	UF : 0, UT : 1,		CONFIG : 'N U T, 0, 0, 0',
	X = 1234.829  mm,	Y = 64.155  mm,	Z = -234.238  mm,
	W = 0.000 deg,	P = 30.000 deg,	R = -177.816 deg
};
P[281]{
   GP1:
	UF : 0, UT : 1,		CONFIG : 'N U T, 0, 0, 0',
	X = 1234.753  mm,	Y = 66.153  mm,	Z = -234.205  mm,
	W = 0.000 deg,	P = 30.000 deg,	R = -177.816 deg
};
P[282]{
   GP1:
	UF : 0, UT : 1,		CONFIG : 'N U T, 0, 0, 0',
	X = 1234.676  mm,	Y = 68.152  mm,	Z = -234.172  mm,
	W = 0.000 deg,	P = 30.000 deg,	R = -177.816 deg
};
P[283]{
   GP1:
	UF : 0, UT : 1,		CONFIG : 'N U T, 0, 0, 0',
	X = 1234.600  mm,	Y = 70.150  mm,	Z = -234.139  mm,
	W = 0.000 deg,	P = 30.000 deg,	R = -177.816 deg
};
P[284]{
   GP1:
	UF : 0, UT : 1,		CONFIG : 'N U T, 0, 0, 0',
	X = 1234.524  mm,	Y = 72.148  mm,	Z = -234.106  mm,
	W = 0.000 deg,	P = 30.000 deg,	R = -177.816 deg
};
P[285]{
   GP1:
	UF : 0, UT : 1,		CONFIG : 'N U T, 0, 0, 0',
	X = 1234.448  mm,	Y = 74.147  mm,	Z = -234.073  mm,
	W = 0.000 deg,	P = 30.000 deg,	R = -172.061 deg
};
P[286]{
   GP1:
	UF : 0, UT : 1,		CONFIG : 'N U T, 0, 0, 0',
	X = 1234.372  mm,	Y = 76.145  mm,	Z = -234.040  mm,
	W = 0.000 deg,	P = 30.000 deg,	R = -168.497 deg
};
P[287]{
   GP1:
	UF : 0, UT : 1,		CONFIG : 'N U T, 0, 0, 0',
	X = 1234.295  mm,	Y = 78.143  mm,	Z = -234.007  mm,
	W = 0.000 deg,	P = 30.000 deg,	R = -164.934 deg
};
P[288]{
   GP1:
	UF : 0, UT : 1,		CONFIG : 'N U T, 0, 0, 0',
	X = 1234.219  mm,	Y = 80.141  mm,	Z = -233.975  mm,
	W = 0.000 deg,	P = 30.000 deg,	R = -161.371 deg
};
P[289]{
   GP1:
	UF : 0, UT : 1,		CONFIG : 'N U T, 0, 0, 0',
	X = 1234.143  mm,	Y = 82.140  mm,	Z = -233.942  mm,
	W = 0.000 deg,	P = 30.000 deg,	R = -160.000 deg
};
P[290]{
   GP1:
	UF : 0, UT : 1,		CONFIG : 'N U T, 0, 0, 0',
	X = 1236.855  mm,	Y = 75.733  mm,	Z = -233.940  mm,
	W = 0.000 deg,	P = 30.000 deg,	R = -160.000 deg
};
P[291]{
   GP1:
	UF : 0, UT : 1,		CONFIG : 'N U T, 0, 0, 0',
	X = 1235.684  mm,	Y = 76.913  mm,	Z = -233.631  mm,
	W = 0.000 deg,	P = 30.000 deg,	R = -160.000 deg
};
P[292]{
   GP1:
	UF : 0, UT : 1,		CONFIG : 'N U T, 0, 0, 0',
	X = 1234.296  mm,	Y = 78.316  mm,	Z = -233.311  mm,
	W = 0.000 deg,	P = 30.000 deg,	R = -160.000 deg
};
P[293]{
   GP1:
	UF : 0, UT : 1,		CONFIG : 'N U T, 0, 0, 0',
	X = 1232.907  mm,	Y = 79.720  mm,	Z = -232.991  mm,
	W = 0.000 deg,	P = 30.000 deg,	R = -160.000 deg
};
P[294]{
   GP1:
	UF : 0, UT : 1,		CONFIG : 'N U T, 0, 0, 0',
	X = 1231.519  mm,	Y = 81.123  mm,	Z = -232.670  mm,
	W = 0.000 deg,	P = 30.000 deg,	R = -160.000 deg
};
P[295]{
   GP1:
	UF : 0, UT : 1,		CONFIG : 'N U T, 0, 0, 0',
	X = 1230.131  mm,	Y = 82.527  mm,	Z = -232.350  mm,
	W = 0.000 deg,	P = 30.000 deg,	R = -160.000 deg
};
P[296]{
   GP1:
	UF : 0, UT : 1,		CONFIG : 'N U T, 0, 0, 0',
	X = 1228.742  mm,	Y = 83.931  mm,	Z = -232.030  mm,
	W = 0.000 deg,	P = 30.000 deg,	R = -160.000 deg
};
P[297]{
   GP1:
	UF : 0, UT : 1,		CONFIG : 'N U T, 0, 0, 0',
	X = 1227.354  mm,	Y = 85.334  mm,	Z = -231.709  mm,
	W = 0.000 deg,	P = 30.000 deg,	R = -160.000 deg
};
P[298]{
   GP1:
	UF : 0, UT : 1,		CONFIG : 'N U T, 0, 0, 0',
	X = 1225.966  mm,	Y = 86.738  mm,	Z = -231.389  mm,
	W = 0.000 deg,	P = 30.000 deg,	R = -160.000 deg
};
P[299]{
   GP1:
	UF : 0, UT : 1,		CONFIG : 'N U T, 0, 0, 0',
	X = 1224.577  mm,	Y = 88.141  mm,	Z = -231.068  mm,
	W = 0.000 deg,	P = 30.000 deg,	R = -160.000 deg
};
P[300]{
   GP1:
	UF : 0, UT : 1,		CONFIG : 'N U T, 0, 0, 0',
	X = 1223.189  mm,	Y = 89.545  mm,	Z = -230.748  mm,
	W = 0.000 deg,	P = 30.000 deg,	R = -160.000 deg
};
P[301]{
   GP1:
	UF : 0, UT : 1,		CONFIG : 'N U T, 0, 0, 0',
	X = 1221.801  mm,	Y = 90.948  mm,	Z = -230.428  mm,
	W = 0.000 deg,	P = 30.000 deg,	R = -160.000 deg
};
P[302]{
   GP1:
	UF : 0, UT : 1,		CONFIG : 'N U T, 0, 0, 0',
	X = 1220.413  mm,	Y = 92.352  mm,	Z = -230.107  mm,
	W = 0.000 deg,	P = 30.000 deg,	R = -160.000 deg
};
P[303]{
   GP1:
	UF : 0, UT : 1,		CONFIG : 'N U T, 0, 0, 0',
	X = 1219.024  mm,	Y = 93.755  mm,	Z = -229.787  mm,
	W = 0.000 deg,	P = 30.000 deg,	R = -160.000 deg
};
P[304]{
   GP1:
	UF : 0, UT : 1,		CONFIG : 'N U T, 0, 0, 0',
	X = 1217.636  mm,	Y = 95.159  mm,	Z = -229.467  mm,
	W = 0.000 deg,	P = 30.000 deg,	R = -160.000 deg
};
P[305]{
   GP1:
	UF : 0, UT : 1,		CONFIG : 'N U T, 0, 0, 0',
	X = 1216.248  mm,	Y = 96.563  mm,	Z = -229.146  mm,
	W = 0.000 deg,	P = 30.000 deg,	R = -160.000 deg
};
P[306]{
   GP1:
	UF : 0, UT : 1,		CONFIG : 'N U T, 0, 0, 0',
	X = 1214.859  mm,	Y = 97.966  mm,	Z = -228.826  mm,
	W = 0.000 deg,	P = 30.000 deg,	R = -160.000 deg
};
P[307]{
   GP1:
	UF : 0, UT : 1,		CONFIG : 'N U T, 0, 0, 0',
	X = 1213.471  mm,	Y = 99.370  mm,	Z = -228.506  mm,
	W = 0.000 deg,	P = 30.000 deg,	R = -160.000 deg
};
P[308]{
   GP1:
	UF : 0, UT : 1,		CONFIG : 'N U T, 0, 0, 0',
	X = 1212.083  mm,	Y = 100.773  mm,	Z = -228.185  mm,
	W = 0.000 deg,	P = 30.000 deg,	R = -160.000 deg
};
P[309]{
   GP1:
	UF : 0, UT : 1,		CONFIG : 'N U T, 0, 0, 0',
	X = 1210.694  mm,	Y = 102.177  mm,	Z = -227.865  mm,
	W = 0.000 deg,	P = 30.000 deg,	R = -160.000 deg
};
P[310]{
   GP1:
	UF : 0, UT : 1,		CONFIG : 'N U T, 0, 0, 0',
	X = 1209.306  mm,	Y = 103.580  mm,	Z = -227.544  mm,
	W = 0.000 deg,	P = 30.000 deg,	R = -160.000 deg
};
P[311]{
   GP1:
	UF : 0, UT : 1,		CONFIG : 'N U T, 0, 0, 0',
	X = 1207.918  mm,	Y = 104.984  mm,	Z = -227.224  mm,
	W = 0.000 deg,	P = 30.000 deg,	R = -160.000 deg
};
P[312]{
   GP1:
	UF : 0, UT : 1,		CONFIG : 'N U T, 0, 0, 0',
	X = 1206.529  mm,	Y = 106.387  mm,	Z = -226.904  mm,
	W = 0.000 deg,	P = 30.000 deg,	R = -168.211 deg
};
P[313]{
   GP1:
	UF : 0, UT : 1,		CONFIG : 'N U T, 0, 0, 0',
	X = 1205.141  mm,	Y = 107.791  mm,	Z = -226.583  mm,
	W = 0.000 deg,	P = 30.000 deg,	R = -172.389 deg
};
P[314]{
   GP1:
	UF : 0, UT : 1,		CONFIG : 'N U T, 0, 0, 0',
	X = 1203.753  mm,	Y = 109.195  mm,	Z = -226.263  mm,
	W = 0.000 deg,	P = 30.000 deg,	R = -176.568 deg
};
P[315]{
   GP1:
	UF : 0, UT : 1,		CONFIG : 'N U T, 0, 0, 0',
	X = 1202.365  mm,	Y = 110.598  mm,	Z = -225.943  mm,
	W = 0.000 deg,	P = 30.000 deg,	R = 179.253 deg
};
P[316]{
   GP1:
	UF : 0, UT : 1,		CONFIG : 'N U T, 0, 0, 0',
	X = 1200.914  mm,	Y = 112.066  mm,	Z = -225.628  mm,
	W = 0.000 deg,	P = 30.000 deg,	R = 179.107 deg
};
P[317]{
   GP1:
	UF : 0, UT : 1,		CONFIG : 'N U T, 0, 0, 0',
	X = 1198.111  mm,	Y = 119.200  mm,	Z = -225.627  mm,
	W = 0.000 deg,	P = 30.000 deg,	R = 179.107 deg
};
P[318]{
   GP1:
	UF : 0, UT : 1,		CONFIG : 'N U T, 0, 0, 0',
	X = 1198.142  mm,	Y = 121.200  mm,	Z = -225.613  mm,
	W = 0.000 deg,	P = 30.000 deg,	R = 179.107 deg
};
P[319]{
   GP1:
	UF : 0, UT : 1,		CONFIG : 'N U T, 0, 0, 0',
	X = 1198.174  mm,	Y = 123.199  mm,	Z = -225.598  mm,
	W = 0.000 deg,	P = 30.000 deg,	R = 179.107 deg
};
P[320]{
   GP1:
	UF : 0, UT : 1,		CONFIG : 'N U T, 0, 0, 0',
	X = 1198.205  mm,	Y = 125.199  mm,	Z = -225.584  mm,
	W = 0.000 deg,	P = 30.000 deg,	R = 179.107 deg
};
P[321]{
   GP1:
	UF : 0, UT : 1,		CONFIG : 'N U T, 0, 0, 0',
	X = 1198.236  mm,	Y = 127.199  mm,	Z = -225.569  mm,
	W = 0.000 deg,	P = 30.000 deg,	R = 179.107 deg
};
P[322]{
   GP1:
	UF : 0, UT : 1,		CONFIG : 'N U T, 0, 0, 0',
	X = 1198.267  mm,	Y = 129.199  mm,	Z = -225.555  mm,
	W = 0.000 deg,	P = 30.000 deg,	R = 179.107 deg
};
P[323]{
   GP1:
	UF : 0, UT : 1,		CONFIG : 'N U T, 0, 0, 0',
	X = 1198.298  mm,	Y = 131.198  mm,	Z = -225.540  mm,
	W = 0.000 deg,	P = 30.000 deg,	R = 179.107 deg
};
P[324]{
   GP1:
	UF : 0, UT : 1,		CONFIG : 'N U T, 0, 0, 0',
	X = 1198.329  mm,	Y = 133.198  mm,	Z = -225.525  mm,
	W = 0.000 deg,	P = 30.000 deg,	R = 179.107 deg
};
P[325]{
   GP1:
	UF : 0, UT : 1,		CONFIG : 'N U T, 0, 0, 0',
	X = 1198.361  mm,	Y = 135.198  mm,	Z = -225.511  mm,
	W = 0.000 deg,	P = 30.000 deg,	R = 179.107 deg
};
P[326]{
   GP1:
	UF : 0, UT : 1,		CONFIG : 'N U T, 0, 0, 0',
	X = 1198.392  mm,	Y = 137.197  mm,	Z = -225.496  mm,
	W = 0.000 deg,	P = 30.000 deg,	R = 179.107 deg
};
P[327]{
   GP1:
	UF : 0, UT : 1,		CONFIG : 'N U T, 0, 0, 0',
	X = 1198.423  mm,	Y = 139.197  mm,	Z = -225.482  mm,
	W = 0.000 deg,	P = 30.000 deg,	R = 179.107 deg
};
P[328]{
   GP1:
	UF : 0, UT : 1,		CONFIG : 'N U T, 0, 0, 0',
	X = 1198.454  mm,	Y = 141.197  mm,	Z = -225.467  mm,
	W = 0.000 deg,	P = 30.000 deg,	R = 179.107 deg
};
P[329]{
   GP1:
	UF : 0, UT : 1,		CONFIG : 'N U T, 0, 0, 0',
	X = 1198.485  mm,	Y = 143.196  mm,	Z = -225.453  mm,
	W = 0.000 deg,	P = 30.000 deg,	R = 179.107 deg
};
P[330]{
   GP1:
	UF : 0, UT : 1,		CONFIG : 'N U T, 0, 0, 0',
	X = 1198.517  mm,	Y = 145.196  mm,	Z = -225.438  mm,
	W = 0.000 deg,	P = 30.000 deg,	R = 179.107 deg
};
P[331]{
   GP1:
	UF : 0, UT : 1,		CONFIG : 'N U T, 0, 0, 0',
	X = 1198.548  mm,	Y = 147.196  mm,	Z = -225.423  mm,
	W = 0.000 deg,	P = 30.000 deg,	R = 179.107 deg
};
P[332]{
   GP1:
	UF : 0, UT : 1,		CONFIG : 'N U T, 0, 0, 0',
	X = 1198.579  mm,	Y = 149.196  mm,	Z = -225.409  mm,
	W = 0.000 deg,	P = 30.000 deg,	R = 179.107 deg
};
P[333]{
   GP1:
	UF : 0, UT : 1,		CONFIG : 'N U T, 0, 0, 0',
	X = 1198.610  mm,	Y = 151.195  mm,	Z = -225.394  mm,
	W = 0.000 deg,	P = 30.000 deg,	R = 179.107 deg
};
P[334]{
   GP1:
	UF : 0, UT : 1,		CONFIG : 'N U T, 0, 0, 0',
	X = 1198.641  mm,	Y = 153.195  mm,	Z = -225.380  mm,
	W = 0.000 deg,	P = 30.000 deg,	R = 179.107 deg
};
P[335]{
   GP1:
	UF : 0, UT : 1,		CONFIG : 'N U T, 0, 0, 0',
	X = 1198.672  mm,	Y = 155.195  mm,	Z = -225.365  mm,
	W = 0.000 deg,	P = 30.000 deg,	R = 179.107 deg
};
P[336]{
   GP1:
	UF : 0, UT : 1,		CONFIG : 'N U T, 0, 0, 0',
	X = 1198.704  mm,	Y = 157.194  mm,	Z = -225.351  mm,
	W = 0.000 deg,	P = 30.000 deg,	R = 179.107 deg
};
P[337]{
   GP1:
	UF : 0, UT : 1,		CONFIG : 'N U T, 0, 0, 0',
	X = 1198.735  mm,	Y = 159.194  mm,	Z = -225.336  mm,
	W = 0.000 deg,	P = 30.000 deg,	R = 179.107 deg
};
P[338]{
   GP1:
	UF : 0, UT : 1,		CONFIG : 'N U T, 0, 0, 0',
	X = 1198.766  mm,	Y = 161.194  mm,	Z = -225.322  mm,
	W = 0.000 deg,	P = 30.000 deg,	R = 179.107 deg
};
P[339]{
   GP1:
	UF : 0, UT : 1,		CONFIG : 'N U T, 0, 0, 0',
	X = 1198.797  mm,	Y = 163.194  mm,	Z = -225.307  mm,
	W = 0.000 deg,	P = 30.000 deg,	R = 179.107 deg
};
P[340]{
   GP1:
	UF : 0, UT : 1,		CONFIG : 'N U T, 0, 0, 0',
	X = 1198.828  mm,	Y = 165.193  mm,	Z = -225.292  mm,
	W = 0.000 deg,	P = 30.000 deg,	R = 179.107 deg
};
P[341]{
   GP1:
	UF : 0, UT : 1,		CONFIG : 'N U T, 0, 0, 0',
	X = 1198.859  mm,	Y = 167.193  mm,	Z = -225.278  mm,
	W = 0.000 deg,	P = 30.000 deg,	R = 179.107 deg
};
P[342]{
   GP1:
	UF : 0, UT : 1,		CONFIG : 'N U T, 0, 0, 0',
	X = 1198.891  mm,	Y = 169.193  mm,	Z = -225.263  mm,
	W = 0.000 deg,	P = 30.000 deg,	R = 179.042 deg
};
P[343]{
   GP1:
	UF : 0, UT : 1,		CONFIG : 'N U T, 0, 0, 0',
	X = 1198.922  mm,	Y = 171.192  mm,	Z = -225.249  mm,
	W = 0.000 deg,	P = 30.000 deg,	R = 175.220 deg
};
P[344]{
   GP1:
	UF : 0, UT : 1,		CONFIG : 'N U T, 0, 0, 0',
	X = 1198.953  mm,	Y = 173.192  mm,	Z = -225.234  mm,
	W = 0.000 deg,	P = 30.000 deg,	R = 171.399 deg
};
P[345]{
   GP1:
	UF : 0, UT : 1,		CONFIG : 'N U T, 0, 0, 0',
	X = 1198.984  mm,	Y = 175.192  mm,	Z = -225.220  mm,
	W = 0.000 deg,	P = 30.000 deg,	R = 167.578 deg
};
P[346]{
   GP1:
	UF : 0, UT : 1,		CONFIG : 'N U T, 0, 0, 0',
	X = 1199.015  mm,	Y = 177.191  mm,	Z = -225.205  mm,
	W = 0.000 deg,	P = 30.000 deg,	R = 163.756 deg
};
P[347]{
   GP1:
	UF : 0, UT : 1,		CONFIG : 'N U T, 0, 0, 0',
	X = 1199.047  mm,	Y = 179.191  mm,	Z = -225.190  mm,
	W = 0.000 deg,	P = 30.000 deg,	R = 160.000 deg
};
P[348]{
   GP1:
	UF : 0, UT : 1,		CONFIG : 'N U T, 0, 0, 0',
	X = 1201.866  mm,	Y = 186.014  mm,	Z = -225.190  mm,
	W = 0.000 deg,	P = 30.000 deg,	R = 160.000 deg
};
P[349]{
   GP1:
	UF : 0, UT : 1,		CONFIG : 'N U T, 0, 0, 0',
	X = 1203.282  mm,	Y = 187.456  mm,	Z = -225.507  mm,
	W = 0.000 deg,	P = 30.000 deg,	R = 160.000 deg
};
P[350]{
   GP1:
	UF : 0, UT : 1,		CONFIG : 'N U T, 0, 0, 0',
	X = 1204.665  mm,	Y = 188.865  mm,	Z = -225.827  mm,
	W = 0.000 deg,	P = 30.000 deg,	R = 160.000 deg
};
P[351]{
   GP1:
	UF : 0, UT : 1,		CONFIG : 'N U T, 0, 0, 0',
	X = 1206.048  mm,	Y = 190.273  mm,	Z = -226.147  mm,
	W = 0.000 deg,	P = 30.000 deg,	R = 160.000 deg
};
P[352]{
   GP1:
	UF : 0, UT : 1,		CONFIG : 'N U T, 0, 0, 0',
	X = 1207.432  mm,	Y = 191.682  mm,	Z = -226.467  mm,
	W = 0.000 deg,	P = 30.000 deg,	R = 160.000 deg
};
P[353]{
   GP1:
	UF : 0, UT : 1,		CONFIG : 'N U T, 0, 0, 0',
	X = 1208.815  mm,	Y = 193.090  mm,	Z = -226.787  mm,
	W = 0.000 deg,	P = 30.000 deg,	R = 160.000 deg
};
P[354]{
   GP1:
	UF : 0, UT : 1,		CONFIG : 'N U T, 0, 0, 0',
	X = 1210.198  mm,	Y = 194.499  mm,	Z = -227.107  mm,
	W = 0.000 deg,	P = 30.000 deg,	R = 160.000 deg
};
P[355]{
   GP1:
	UF : 0, UT : 1,		CONFIG : 'N U T, 0, 0, 0',
	X = 1211.582  mm,	Y = 195.907  mm,	Z = -227.427  mm,
	W = 0.000 deg,	P = 30.000 deg,	R = 160.000 deg
};
P[356]{
   GP1:
	UF : 0, UT : 1,		CONFIG : 'N U T, 0, 0, 0',
	X = 1212.965  mm,	Y = 197.316  mm,	Z = -227.747  mm,
	W = 0.000 deg,	P = 30.000 deg,	R = 160.000 deg
};
P[357]{
   GP1:
	UF : 0, UT : 1,		CONFIG : 'N U T, 0, 0, 0',
	X = 1214.348  mm,	Y = 198.725  mm,	Z = -228.067  mm,
	W = 0.000 deg,	P = 30.000 deg,	R = 160.000 deg
};
P[358]{
   GP1:
	UF : 0, UT : 1,		CONFIG : 'N U T, 0, 0, 0',
	X = 1215.732  mm,	Y = 200.133  mm,	Z = -228.387  mm,
	W = 0.000 deg,	P = 30.000 deg,	R = 160.000 deg
};
P[359]{
   GP1:
	UF : 0, UT : 1,		CONFIG : 'N U T, 0, 0, 0',
	X = 1217.115  mm,	Y = 201.542  mm,	Z = -228.707  mm,
	W = 0.000 deg,	P = 30.000 deg,	R = 160.000 deg
};
P[360]{
   GP1:
	UF : 0, UT : 1,		CONFIG : 'N U T, 0, 0, 0',
	X = 1218.498  mm,	Y = 202.950  mm,	Z = -229.026  mm,
	W = 0.000 deg,	P = 30.000 deg,	R = 160.000 deg
};
P[361]{
   GP1:
	UF : 0, UT : 1,		CONFIG : 'N U T, 0, 0, 0',
	X = 1219.882  mm,	Y = 204.359  mm,	Z = -229.346  mm,
	W = 0.000 deg,	P = 30.000 deg,	R = 160.000 deg
};
P[362]{
   GP1:
	UF : 0, UT : 1,		CONFIG : 'N U T, 0, 0, 0',
	X = 1221.265  mm,	Y = 205.767  mm,	Z = -229.666  mm,
	W = 0.000 deg,	P = 30.000 deg,	R = 160.000 deg
};
P[363]{
   GP1:
	UF : 0, UT : 1,		CONFIG : 'N U T, 0, 0, 0',
	X = 1222.649  mm,	Y = 207.176  mm,	Z = -229.986  mm,
	W = 0.000 deg,	P = 30.000 deg,	R = 160.000 deg
};
P[364]{
   GP1:
	UF : 0, UT : 1,		CONFIG : 'N U T, 0, 0, 0',
	X = 1224.032  mm,	Y = 208.584  mm,	Z = -230.306  mm,
	W = 0.000 deg,	P = 30.000 deg,	R = 160.000 deg
};
P[365]{
   GP1:
	UF : 0, UT : 1,		CONFIG : 'N U T, 0, 0, 0',
	X = 1225.415  mm,	Y = 209.993  mm,	Z = -230.626  mm,
	W = 0.000 deg,	P = 30.000 deg,	R = 160.000 deg
};
P[366]{
   GP1:
	UF : 0, UT : 1,		CONFIG : 'N U T, 0, 0, 0',
	X = 1226.799  mm,	Y = 211.401  mm,	Z = -230.946  mm,
	W = 0.000 deg,	P = 30.000 deg,	R = 160.000 deg
};
P[367]{
   GP1:
	UF : 0, UT : 1,		CONFIG : 'N U T, 0, 0, 0',
	X = 1228.182  mm,	Y = 212.810  mm,	Z = -231.266  mm,
	W = 0.000 deg,	P = 30.000 deg,	R = 160.000 deg
};
P[368]{
   GP1:
	UF : 0, UT : 1,		CONFIG : 'N U T, 0, 0, 0',
	X = 1229.565  mm,	Y = 214.218  mm,	Z = -231.586  mm,
	W = 0.000 deg,	P = 30.000 deg,	R = 163.943 deg
};
P[369]{
   GP1:
	UF : 0, UT : 1,		CONFIG : 'N U T, 0, 0, 0',
	X = 1230.949  mm,	Y = 215.627  mm,	Z = -231.906  mm,
	W = 0.000 deg,	P = 30.000 deg,	R = 167.922 deg
};
P[370]{
   GP1:
	UF : 0, UT : 1,		CONFIG : 'N U T, 0, 0, 0',
	X = 1232.332  mm,	Y = 217.036  mm,	Z = -232.226  mm,
	W = 0.000 deg,	P = 30.000 deg,	R = 171.902 deg
};
P[371]{
   GP1:
	UF : 0, UT : 1,		CONFIG : 'N U T, 0, 0, 0',
	X = 1233.715  mm,	Y = 218.444  mm,	Z = -232.546  mm,
	W = 0.000 deg,	P = 30.000 deg,	R = 175.881 deg
};
P[372]{
   GP1:
	UF : 0, UT : 1,		CONFIG : 'N U T, 0, 0, 0',
	X = 1235.099  mm,	Y = 219.853  mm,	Z = -232.866  mm,
	W = 0.000 deg,	P = 30.000 deg,	R = 179.860 deg
};
P[373]{
   GP1:
	UF : 0, UT : 1,		CONFIG : 'N U T, 0, 0, 0',
	X = 1234.773  mm,	Y = 219.199  mm,	Z = -233.096  mm,
	W = 0.000 deg,	P = 30.000 deg,	R = 179.897 deg
};
P[374]{
   GP1:
	UF : 0, UT : 1,		CONFIG : 'N U T, 0, 0, 0',
	X = 1233.228  mm,	Y = 214.439  mm,	Z = -233.096  mm,
	W = 0.000 deg,	P = 30.000 deg,	R = 179.897 deg
};
P[375]{
   GP1:
	UF : 0, UT : 1,		CONFIG : 'N U T, 0, 0, 0',
	X = 1233.232  mm,	Y = 216.439  mm,	Z = -233.096  mm,
	W = 0.000 deg,	P = 30.000 deg,	R = 179.897 deg
};
P[376]{
   GP1:
	UF : 0, UT : 1,		CONFIG : 'N U T, 0, 0, 0',
	X = 1233.235  mm,	Y = 218.439  mm,	Z = -233.096  mm,
	W = 0.000 deg,	P = 30.000 deg,	R = 179.897 deg
};
P[377]{
   GP1:
	UF : 0, UT : 1,		CONFIG : 'N U T, 0, 0, 0',
	X = 1233.239  mm,	Y = 220.439  mm,	Z = -233.097  mm,
	W = 0.000 deg,	P = 30.000 deg,	R = 179.897 deg
};
P[378]{
   GP1:
	UF : 0, UT : 1,		CONFIG : 'N U T, 0, 0, 0',
	X = 1233.243  mm,	Y = 222.439  mm,	Z = -233.097  mm,
	W = 0.000 deg,	P = 30.000 deg,	R = 179.897 deg
};
P[379]{
   GP1:
	UF : 0, UT : 1,		CONFIG : 'N U T, 0, 0, 0',
	X = 1233.246  mm,	Y = 224.439  mm,	Z = -233.097  mm,
	W = 0.000 deg,	P = 30.000 deg,	R = 179.897 deg
};
P[380]{
   GP1:
	UF : 0, UT : 1,		CONFIG : 'N U T, 0, 0, 0',
	X = 1233.249  mm,	Y = 225.876  mm,	Z = -233.098  mm,
	W = 0.000 deg,	P = 30.000 deg,	R = 179.897 deg
};
/END
